C03648=1126.143,285.220,-74.172,-178.101,10.292,149.548
C03649=1126.148,284.972,-74.142,-178.104,10.290,149.548
C03650=1126.152,284.724,-74.112,-178.107,10.287,149.548
C03651=1126.156,284.475,-74.081,-178.109,10.284,149.548
C03652=1126.160,284.228,-74.051,-178.113,10.282,149.549
C03653=1126.165,283.980,-74.020,-178.116,10.279,149.549
C03654=1126.169,283.732,-73.989,-178.119,10.277,149.549
C03655=1126.173,283.483,-73.959,-178.122,10.274,149.549
C03656=1126.177,283.235,-73.928,-178.125,10.272,149.549
C03657=1126.181,282.988,-73.898,-178.128,10.269,149.549
C03658=1126.186,282.739,-73.868,-178.131,10.267,149.549
C03659=1126.189,282.491,-73.837,-178.134,10.265,149.550
C03660=1126.194,282.243,-73.807,-178.137,10.262,149.550
C03661=1126.199,281.995,-73.776,-178.140,10.259,149.550
C03662=1126.202,281.747,-73.746,-178.143,10.257,149.550
C03663=1126.207,281.498,-73.715,-178.146,10.254,149.550
C03664=1126.210,281.285,-73.689,-178.149,10.251,149.551
C03665=1126.214,281.072,-73.663,-178.152,10.249,149.551
C03666=1126.218,280.859,-73.638,-178.155,10.247,149.551
C03667=1126.221,280.645,-73.611,-178.158,10.244,149.551
C03668=1126.224,280.432,-73.585,-178.161,10.242,149.551
C03669=1126.228,280.218,-73.559,-178.164,10.239,149.551
C03670=1126.232,280.006,-73.533,-178.167,10.237,149.552
C03671=1126.235,279.791,-73.507,-178.170,10.235,149.552
C03672=1126.239,279.543,-73.477,-178.173,10.232,149.552
C03673=1126.244,279.295,-73.446,-178.177,10.229,149.552
C03674=1126.248,279.047,-73.417,-178.180,10.226,149.553
C03675=1126.253,278.799,-73.386,-178.183,10.224,149.553
C03676=1126.256,278.550,-73.356,-178.187,10.221,149.553
C03677=1126.260,278.303,-73.326,-178.190,10.218,149.553
C03678=1126.265,278.055,-73.295,-178.193,10.215,149.553
C03679=1126.269,277.806,-73.266,-178.196,10.212,149.553
C03680=1126.273,277.559,-73.236,-178.200,10.210,149.554
C03681=1126.278,277.310,-73.206,-178.203,10.207,149.554
C03682=1126.282,277.063,-73.175,-178.206,10.204,149.554
C03683=1126.285,276.814,-73.146,-178.210,10.201,149.554
C03684=1126.290,276.565,-73.115,-178.213,10.199,149.554
C03685=1126.294,276.317,-73.085,-178.215,10.196,149.554
C03686=1126.298,276.069,-73.056,-178.219,10.193,149.555
C03687=1126.302,275.821,-73.026,-178.222,10.191,149.555
C03688=1126.307,275.573,-72.996,-178.225,10.188,149.555
C03689=1126.311,275.325,-72.965,-178.228,10.185,149.555
C03690=1126.315,275.077,-72.936,-178.232,10.182,149.555
C03691=1126.319,274.829,-72.907,-178.235,10.179,149.555
C03692=1126.324,274.581,-72.876,-178.237,10.176,149.555
C03693=1126.328,274.332,-72.846,-178.241,10.174,149.556
C03694=1126.332,274.084,-72.817,-178.244,10.171,149.556
C03695=1126.335,273.836,-72.786,-178.247,10.168,149.556
C03696=1126.340,273.587,-72.756,-178.250,10.166,149.556
C03697=1126.345,273.339,-72.727,-178.253,10.163,149.556
C03698=1126.349,273.091,-72.697,-178.256,10.160,149.556
C03699=1126.353,272.843,-72.667,-178.258,10.159,149.556
C03700=1126.357,272.595,-72.638,-178.261,10.156,149.557
C03701=1126.361,272.347,-72.608,-178.264,10.153,149.557
C03702=1126.366,272.098,-72.578,-178.267,10.150,149.557
C03703=1126.370,271.850,-72.549,-178.270,10.148,149.557
C03704=1126.374,271.602,-72.519,-178.273,10.145,149.557
C03705=1126.378,271.354,-72.489,-178.276,10.142,149.557
C03706=1126.382,271.106,-72.460,-178.279,10.139,149.557
C03707=1126.387,270.857,-72.430,-178.281,10.137,149.557
C03708=1126.391,270.609,-72.401,-178.284,10.134,149.557
C03709=1126.395,270.361,-72.371,-178.287,10.132,149.558
C03710=1126.399,270.112,-72.342,-178.290,10.129,149.558
C03711=1126.403,269.864,-72.312,-178.292,10.127,149.558
C03712=1126.409,269.616,-72.283,-178.295,10.124,149.558
C03713=1126.413,269.368,-72.253,-178.298,10.121,149.558
C03714=1126.417,269.120,-72.223,-178.301,10.119,149.558
C03715=1126.421,268.872,-72.194,-178.303,10.117,149.558
C03716=1126.425,268.624,-72.164,-178.306,10.114,149.558
C03717=1126.429,268.376,-72.135,-178.309,10.111,149.558
C03718=1126.434,268.127,-72.105,-178.312,10.109,149.558
C03719=1126.438,267.879,-72.076,-178.314,10.106,149.559
C03720=1126.441,267.666,-72.051,-178.317,10.105,149.559
C03721=1126.445,267.452,-72.026,-178.319,10.102,149.559
C03722=1126.449,267.238,-72.001,-178.321,10.100,149.559
C03723=1126.452,267.025,-71.976,-178.323,10.098,149.559
C03724=1126.456,266.811,-71.951,-178.326,10.096,149.559
C03725=1126.460,266.598,-71.925,-178.328,10.094,149.559
C03726=1126.464,266.384,-71.900,-178.330,10.092,149.559
C03727=1126.467,266.171,-71.875,-178.332,10.090,149.559
C03728=1126.471,265.922,-71.845,-178.335,10.087,149.559
C03729=1126.476,265.674,-71.816,-178.337,10.085,149.559
C03730=1126.480,265.426,-71.786,-178.340,10.083,149.560
C03731=1126.484,265.178,-71.757,-178.343,10.080,149.560
C03732=1126.489,264.929,-71.728,-178.345,10.078,149.560
C03733=1126.492,264.681,-71.699,-178.347,10.075,149.560
C03734=1126.497,264.433,-71.670,-178.350,10.073,149.560
C03735=1126.501,264.185,-71.641,-178.354,10.070,149.560
C03736=1126.505,263.937,-71.611,-178.358,10.067,149.560
C03737=1126.510,263.688,-71.582,-178.362,10.064,149.561
C03738=1126.514,263.440,-71.553,-178.365,10.061,149.561
C03739=1126.518,263.191,-71.524,-178.369,10.058,149.561
C03740=1126.523,262.944,-71.494,-178.373,10.055,149.561
C03741=1126.527,262.695,-71.466,-178.376,10.052,149.561
C03742=1126.531,262.447,-71.437,-178.380,10.049,149.562
C03743=1126.535,262.199,-71.407,-178.383,10.045,149.562
C03744=1126.539,261.950,-71.379,-178.387,10.043,149.562
C03745=1126.544,261.702,-71.350,-178.390,10.039,149.562
C03746=1126.548,261.454,-71.321,-178.393,10.037,149.563
C03747=1126.552,261.205,-71.292,-178.397,10.033,149.563
C03748=1126.556,260.957,-71.263,-178.400,10.031,149.563
C03749=1126.561,260.709,-71.234,-178.404,10.027,149.563
C03750=1126.565,260.461,-71.205,-178.407,10.025,149.563
C03751=1126.569,260.212,-71.177,-178.410,10.021,149.563
C03752=1126.573,259.964,-71.147,-178.413,10.018,149.563
C03753=1126.579,259.716,-71.119,-178.416,10.016,149.563
C03754=1126.582,259.468,-71.090,-178.420,10.012,149.564
C03755=1126.586,259.219,-71.061,-178.423,10.010,149.564
C03756=1126.591,258.970,-71.032,-178.426,10.007,149.564
C03757=1126.595,258.723,-71.004,-178.429,10.004,149.564
C03758=1126.599,258.474,-70.974,-178.433,10.001,149.564
C03759=1126.604,258.225,-70.946,-178.436,9.998,149.564
C03760=1126.608,257.978,-70.918,-178.439,9.995,149.564
C03761=1126.612,257.729,-70.888,-178.442,9.992,149.564
C03762=1126.616,257.481,-70.860,-178.444,9.990,149.565
C03763=1126.621,257.233,-70.832,-178.448,9.986,149.564
C03764=1126.625,256.984,-70.802,-178.451,9.983,149.565
C03765=1126.629,256.736,-70.774,-178.454,9.980,149.565
C03766=1126.634,256.487,-70.746,-178.456,9.978,149.565
C03767=1126.638,256.240,-70.717,-178.459,9.975,149.565
C03768=1126.642,255.991,-70.688,-178.462,9.972,149.565
C03769=1126.646,255.743,-70.661,-178.462,9.971,149.565
C03770=1126.651,255.495,-70.631,-178.462,9.970,149.564
C03771=1126.655,255.246,-70.602,-178.462,9.969,149.564
C03772=1126.659,254.998,-70.575,-178.462,9.968,149.564
C03773=1126.664,254.749,-70.546,-178.462,9.967,149.564
C03774=1126.668,254.502,-70.517,-178.463,9.966,149.564
C03775=1126.672,254.253,-70.489,-178.464,9.964,149.563
C03776=1126.676,254.039,-70.464,-178.465,9.963,149.563
C03777=1126.679,253.826,-70.440,-178.466,9.962,149.563
C03778=1126.683,253.612,-70.415,-178.467,9.960,149.563
C03779=1126.687,253.397,-70.391,-178.468,9.959,149.563
C03780=1126.691,253.185,-70.366,-178.471,9.957,149.563
C03781=1126.694,252.971,-70.342,-178.472,9.955,149.563
C03782=1126.698,252.757,-70.318,-178.474,9.953,149.564
C03783=1126.702,252.544,-70.292,-178.476,9.951,149.564
C03784=1126.706,252.296,-70.265,-178.479,9.949,149.564
C03785=1126.710,252.047,-70.236,-178.482,9.946,149.564
C03786=1126.714,251.798,-70.208,-178.485,9.944,149.564
C03787=1126.719,251.550,-70.179,-178.488,9.941,149.564
C03788=1126.723,251.301,-70.151,-178.492,9.938,149.565
C03789=1126.728,251.054,-70.122,-178.495,9.936,149.565
C03790=1126.732,250.805,-70.094,-178.499,9.933,149.565
C03791=1126.736,250.556,-70.065,-178.504,9.929,149.566
C03792=1126.740,250.309,-70.037,-178.508,9.925,149.566
C03793=1126.745,250.060,-70.009,-178.513,9.922,149.566
C03794=1126.749,249.812,-69.981,-178.518,9.918,149.567
C03795=1126.753,249.563,-69.953,-178.523,9.914,149.567
C03796=1126.758,249.315,-69.924,-178.528,9.911,149.568
C03797=1126.762,249.066,-69.896,-178.533,9.906,149.568
C03798=1126.766,248.819,-69.868,-178.539,9.902,149.568
C03799=1126.771,248.570,-69.840,-178.545,9.896,149.569
C03800=1126.775,248.322,-69.812,-178.551,9.892,149.569
C03801=1126.779,248.073,-69.785,-178.557,9.887,149.570
C03802=1126.784,247.824,-69.756,-178.564,9.882,149.570
C03803=1126.788,247.576,-69.728,-178.570,9.877,149.571
C03804=1126.792,247.328,-69.700,-178.575,9.873,149.571
C03805=1126.796,247.079,-69.672,-178.576,9.870,149.571
C03806=1126.801,246.831,-69.645,-178.577,9.869,149.571
C03807=1126.806,246.583,-69.617,-178.579,9.866,149.570
C03808=1126.809,246.334,-69.589,-178.580,9.865,149.570
C03809=1126.814,246.086,-69.561,-178.582,9.862,149.570
C03810=1126.818,245.837,-69.533,-178.583,9.860,149.570
C03811=1126.822,245.589,-69.506,-178.585,9.858,149.570
C03812=1126.827,245.340,-69.477,-178.586,9.855,149.570
C03813=1126.831,245.092,-69.450,-178.588,9.853,149.570
C03814=1126.836,244.844,-69.422,-178.589,9.851,149.570
C03815=1126.839,244.595,-69.394,-178.591,9.849,149.570
C03816=1126.844,244.347,-69.367,-178.593,9.846,149.569
C03817=1126.849,244.098,-69.338,-178.595,9.844,149.569
C03818=1126.853,243.850,-69.310,-178.597,9.842,149.569
C03819=1126.858,243.602,-69.283,-178.598,9.839,149.569
C03820=1126.861,243.353,-69.255,-178.600,9.837,149.569
C03821=1126.866,243.105,-69.227,-178.602,9.836,149.569
C03822=1126.870,242.857,-69.200,-178.604,9.834,149.569
C03823=1126.874,242.608,-69.172,-178.606,9.831,149.569
C03824=1126.879,242.360,-69.145,-178.608,9.828,149.569
C03825=1126.883,242.111,-69.116,-178.610,9.826,149.569
C03826=1126.888,241.862,-69.089,-178.612,9.823,149.569
C03827=1126.892,241.614,-69.061,-178.614,9.821,149.569
C03828=1126.896,241.366,-69.033,-178.616,9.819,149.569
C03829=1126.901,241.117,-69.006,-178.618,9.817,149.569
C03830=1126.905,240.869,-68.978,-178.621,9.815,149.569
C03831=1126.909,240.620,-68.951,-178.623,9.812,149.569
C03832=1126.913,240.407,-68.928,-178.625,9.810,149.569
C03833=1126.917,240.192,-68.904,-178.627,9.808,149.569
C03834=1126.921,239.979,-68.880,-178.629,9.806,149.569
C03835=1126.924,239.766,-68.856,-178.631,9.804,149.569
C03836=1126.928,239.551,-68.833,-178.633,9.802,149.569
C03837=1126.932,239.338,-68.809,-178.635,9.800,149.569
C03838=1126.936,239.124,-68.785,-178.637,9.797,149.569
C03839=1126.940,238.910,-68.762,-178.639,9.795,149.569
C03840=1126.943,238.662,-68.734,-178.642,9.793,149.569
C03841=1126.948,238.413,-68.707,-178.644,9.790,149.569
C03842=1126.952,238.165,-68.679,-178.647,9.787,149.570
C03843=1126.957,237.916,-68.651,-178.649,9.785,149.570
C03844=1126.961,237.668,-68.624,-178.652,9.783,149.570
C03845=1126.966,237.420,-68.597,-178.655,9.780,149.570
C03846=1126.970,237.171,-68.570,-178.657,9.778,149.570
C03847=1126.974,236.922,-68.542,-178.660,9.775,149.570
C03848=1126.979,236.674,-68.514,-178.663,9.772,149.570
C03849=1126.983,236.426,-68.487,-178.666,9.769,149.570
C03850=1126.987,236.177,-68.460,-178.669,9.767,149.570
C03851=1126.991,235.929,-68.433,-178.672,9.764,149.570
C03852=1126.996,235.681,-68.406,-178.674,9.761,149.570
C03853=1127.000,235.432,-68.379,-178.677,9.758,149.571
C03854=1127.005,235.184,-68.352,-178.680,9.755,149.571
C03855=1127.009,234.935,-68.323,-178.683,9.753,149.571
C03856=1127.013,234.686,-68.296,-178.686,9.750,149.571
C03857=1127.018,234.438,-68.269,-178.689,9.747,149.571
C03858=1127.022,234.190,-68.243,-178.692,9.744,149.571
C03859=1127.026,233.941,-68.215,-178.695,9.742,149.571
C03860=1127.030,233.693,-68.188,-178.699,9.738,149.572
C03861=1127.035,233.444,-68.161,-178.702,9.736,149.572
C03862=1127.040,233.196,-68.133,-178.705,9.733,149.572
C03863=1127.044,232.947,-68.106,-178.709,9.729,149.572
C03864=1127.048,232.699,-68.080,-178.711,9.727,149.572
C03865=1127.052,232.450,-68.053,-178.714,9.724,149.572
C03866=1127.057,232.201,-68.025,-178.718,9.720,149.572
C03867=1127.062,231.953,-67.998,-178.721,9.718,149.572
C03868=1127.065,231.705,-67.972,-178.725,9.714,149.573
C03869=1127.070,231.456,-67.945,-178.728,9.711,149.573
C03870=1127.075,231.208,-67.918,-178.731,9.708,149.573
C03871=1127.079,230.959,-67.891,-178.735,9.705,149.573
C03872=1127.083,230.710,-67.864,-178.739,9.701,149.573
C03873=1127.087,230.462,-67.837,-178.742,9.698,149.573
C03874=1127.092,230.213,-67.810,-178.745,9.695,149.573
C03875=1127.096,229.965,-67.783,-178.749,9.691,149.574
C03876=1127.101,229.717,-67.756,-178.753,9.688,149.574
C03877=1127.105,229.468,-67.729,-178.756,9.685,149.574
C03878=1127.109,229.220,-67.703,-178.760,9.681,149.574
C03879=1127.114,228.971,-67.676,-178.763,9.678,149.574
C03880=1127.119,228.722,-67.649,-178.767,9.674,149.574
C03881=1127.123,228.474,-67.623,-178.771,9.671,149.574
C03882=1127.127,228.226,-67.596,-178.774,9.667,149.575
C03883=1127.131,227.977,-67.569,-178.777,9.664,149.575
C03884=1127.136,227.728,-67.543,-178.781,9.661,149.575
C03885=1127.140,227.479,-67.516,-178.784,9.657,149.575
C03886=1127.144,227.231,-67.489,-178.788,9.653,149.575
C03887=1127.149,226.982,-67.462,-178.790,9.651,149.575
C03888=1127.153,226.769,-67.439,-178.793,9.648,149.575
C03889=1127.157,226.555,-67.416,-178.796,9.645,149.575
C03890=1127.160,226.341,-67.393,-178.799,9.642,149.575
C03891=1127.164,226.127,-67.371,-178.801,9.639,149.575
C03892=1127.168,225.913,-67.349,-178.804,9.636,149.575
C03893=1127.172,225.699,-67.326,-178.807,9.633,149.575
C03894=1127.176,225.485,-67.303,-178.810,9.630,149.575
C03895=1127.180,225.272,-67.280,-178.812,9.627,149.575
C03896=1127.184,225.023,-67.253,-178.816,9.624,149.575
C03897=1127.188,224.774,-67.227,-178.818,9.621,149.575
C03898=1127.192,224.526,-67.201,-178.822,9.617,149.575
C03899=1127.197,224.278,-67.174,-178.825,9.614,149.575
C03900=1127.201,224.029,-67.148,-178.827,9.611,149.575
C03901=1127.206,223.780,-67.121,-178.831,9.607,149.575
C03902=1127.210,223.531,-67.095,-178.833,9.604,149.575
C03903=1127.215,223.283,-67.068,-178.836,9.600,149.575
C03904=1127.219,223.034,-67.043,-178.839,9.597,149.575
C03905=1127.223,222.786,-67.016,-178.842,9.595,149.575
C03906=1127.228,222.537,-66.990,-178.844,9.591,149.575
C03907=1127.232,222.288,-66.964,-178.848,9.588,149.575
C03908=1127.237,222.041,-66.938,-178.850,9.584,149.575
C03909=1127.242,221.791,-66.912,-178.853,9.581,149.575
C03910=1127.246,221.543,-66.885,-178.855,9.578,149.575
C03911=1127.251,221.294,-66.859,-178.858,9.575,149.575
C03912=1127.255,221.045,-66.833,-178.860,9.572,149.575
C03913=1127.259,220.797,-66.807,-178.863,9.568,149.575
C03914=1127.263,220.548,-66.781,-178.866,9.565,149.575
C03915=1127.268,220.300,-66.755,-178.868,9.562,149.575
C03916=1127.272,220.052,-66.728,-178.871,9.559,149.575
C03917=1127.277,219.803,-66.703,-178.873,9.556,149.575
C03918=1127.282,219.554,-66.676,-178.876,9.553,149.575
C03919=1127.285,219.306,-66.650,-178.878,9.550,149.574
C03920=1127.290,219.057,-66.624,-178.880,9.547,149.574
C03921=1127.294,218.808,-66.598,-178.883,9.544,149.574
C03922=1127.299,218.560,-66.572,-178.885,9.541,149.574
C03923=1127.303,218.311,-66.546,-178.888,9.537,149.574
C03924=1127.308,218.063,-66.520,-178.890,9.534,149.574
C03925=1127.312,217.814,-66.494,-178.892,9.532,149.574
C03926=1127.316,217.565,-66.469,-178.894,9.529,149.574
C03927=1127.322,217.317,-66.443,-178.897,9.525,149.574
C03928=1127.326,217.068,-66.416,-178.898,9.523,149.573
C03929=1127.330,216.820,-66.390,-178.901,9.520,149.573
C03930=1127.334,216.571,-66.365,-178.903,9.516,149.573
C03931=1127.338,216.322,-66.339,-178.905,9.514,149.573
C03932=1127.343,216.074,-66.313,-178.907,9.511,149.573
C03933=1127.348,215.825,-66.287,-178.909,9.508,149.573
C03934=1127.352,215.576,-66.261,-178.911,9.505,149.573
C03935=1127.356,215.327,-66.236,-178.913,9.503,149.573
C03936=1127.361,215.079,-66.210,-178.915,9.500,149.572
C03937=1127.366,214.830,-66.184,-178.917,9.497,149.572
C03938=1127.369,214.582,-66.158,-178.919,9.494,149.572
C03939=1127.374,214.333,-66.132,-178.921,9.491,149.572
C03940=1127.378,214.085,-66.107,-178.923,9.488,149.572
C03941=1127.383,213.836,-66.081,-178.924,9.486,149.572
C03942=1127.388,213.587,-66.055,-178.926,9.484,149.572
C03943=1127.392,213.338,-66.029,-178.928,9.481,149.571
C03944=1127.396,213.124,-66.008,-178.930,9.479,149.571
C03945=1127.400,212.910,-65.985,-178.931,9.476,149.571
C03946=1127.403,212.697,-65.963,-178.932,9.474,149.571
C03947=1127.407,212.483,-65.941,-178.934,9.472,149.571
C03948=1127.411,212.269,-65.920,-178.936,9.469,149.571
C03949=1127.415,212.055,-65.897,-178.938,9.467,149.571
C03950=1127.418,211.840,-65.875,-178.939,9.465,149.571
C03951=1127.423,211.626,-65.853,-178.940,9.463,149.570
C03952=1127.427,211.378,-65.828,-178.942,9.460,149.570
C03953=1127.432,211.129,-65.802,-178.945,9.457,149.570
C03954=1127.436,210.880,-65.776,-178.947,9.455,149.570
C03955=1127.441,210.632,-65.751,-178.949,9.453,149.570
C03956=1127.445,210.383,-65.725,-178.951,9.449,149.570
C03957=1127.449,210.135,-65.699,-178.953,9.447,149.570
C03958=1127.454,209.886,-65.675,-178.955,9.445,149.570
C03959=1127.458,209.637,-65.649,-178.957,9.442,149.570
C03960=1127.463,209.388,-65.623,-178.959,9.439,149.570
C03961=1127.467,209.140,-65.598,-178.962,9.436,149.570
C03962=1127.472,208.891,-65.572,-178.964,9.434,149.570
C03963=1127.476,208.643,-65.546,-178.967,9.431,149.570
C03964=1127.481,208.394,-65.522,-178.969,9.428,149.570
C03965=1127.485,208.145,-65.496,-178.972,9.426,149.570
C03966=1127.489,207.896,-65.470,-178.974,9.423,149.570
C03967=1127.494,207.648,-65.445,-178.977,9.420,149.570
C03968=1127.499,207.399,-65.420,-178.979,9.418,149.570
C03969=1127.503,207.151,-65.395,-178.981,9.415,149.570
C03970=1127.507,206.902,-65.369,-178.984,9.412,149.570
C03971=1127.511,206.653,-65.343,-178.987,9.409,149.570
C03972=1127.517,206.405,-65.319,-178.989,9.407,149.570
C03973=1127.521,206.156,-65.293,-178.992,9.404,149.571
C03974=1127.526,205.908,-65.268,-178.995,9.401,149.571
C03975=1127.530,205.658,-65.242,-178.998,9.398,149.571
C03976=1127.535,205.410,-65.217,-179.001,9.396,149.571
C03977=1127.539,205.161,-65.193,-179.003,9.393,149.571
C03978=1127.543,204.912,-65.167,-179.006,9.390,149.571
C03979=1127.548,204.664,-65.142,-179.009,9.387,149.571
C03980=1127.552,204.415,-65.116,-179.012,9.384,149.571
C03981=1127.557,204.167,-65.091,-179.016,9.381,149.571
C03982=1127.562,203.917,-65.066,-179.018,9.378,149.571
C03983=1127.566,203.669,-65.041,-179.021,9.375,149.571
C03984=1127.570,203.420,-65.016,-179.024,9.372,149.572
C03985=1127.575,203.172,-64.991,-179.028,9.369,149.572
C03986=1127.580,202.922,-64.966,-179.031,9.366,149.572
C03987=1127.584,202.675,-64.941,-179.034,9.363,149.572
C03988=1127.588,202.425,-64.916,-179.037,9.360,149.572
C03989=1127.593,202.177,-64.891,-179.040,9.357,149.572
C03990=1127.597,201.928,-64.866,-179.044,9.353,149.572
C03991=1127.602,201.680,-64.841,-179.046,9.350,149.572
C03992=1127.606,201.430,-64.816,-179.050,9.347,149.573
C03993=1127.611,201.182,-64.792,-179.053,9.344,149.573
C03994=1127.615,200.933,-64.766,-179.056,9.341,149.573
C03995=1127.620,200.685,-64.741,-179.060,9.337,149.573
C03996=1127.623,200.436,-64.716,-179.063,9.334,149.573
C03997=1127.629,200.187,-64.691,-179.066,9.331,149.573
C03998=1127.633,199.938,-64.666,-179.070,9.327,149.573
C03999=1127.638,199.689,-64.642,-179.074,9.324,149.573
C04000=1127.641,199.476,-64.621,-179.077,9.321,149.574
C04001=1127.645,199.261,-64.599,-179.080,9.318,149.574
C04002=1127.649,199.047,-64.577,-179.083,9.315,149.574
C04003=1127.653,198.833,-64.557,-179.086,9.312,149.574
C04004=1127.657,198.619,-64.535,-179.089,9.309,149.574
C04005=1127.661,198.405,-64.515,-179.093,9.306,149.574
C04006=1127.665,198.191,-64.493,-179.095,9.303,149.574
C04007=1127.668,197.977,-64.472,-179.099,9.299,149.574
C04008=1127.673,197.728,-64.447,-179.102,9.296,149.575
C04009=1127.677,197.479,-64.423,-179.106,9.292,149.575
C04010=1127.682,197.230,-64.398,-179.109,9.289,149.575
C04011=1127.686,196.981,-64.373,-179.114,9.284,149.575
C04012=1127.691,196.733,-64.349,-179.117,9.281,149.575
C04013=1127.696,196.484,-64.325,-179.121,9.277,149.575
C04014=1127.700,196.235,-64.300,-179.125,9.273,149.575
C04015=1127.705,195.986,-64.276,-179.126,9.271,149.575
C04016=1127.710,195.738,-64.251,-179.127,9.268,149.575
C04017=1127.713,195.489,-64.226,-179.129,9.266,149.575
C04018=1127.718,195.240,-64.201,-179.131,9.263,149.575
C04019=1127.723,194.992,-64.177,-179.132,9.261,149.574
C04020=1127.727,194.743,-64.153,-179.134,9.258,149.574
C04021=1127.732,194.493,-64.129,-179.136,9.256,149.574
C04022=1127.736,194.245,-64.105,-179.137,9.253,149.574
C04023=1127.742,193.996,-64.080,-179.139,9.251,149.574
C04024=1127.745,193.747,-64.055,-179.141,9.248,149.574
C04025=1127.750,193.499,-64.031,-179.142,9.246,149.574
C04026=1127.755,193.250,-64.007,-179.145,9.242,149.574
C04027=1127.759,193.001,-63.982,-179.146,9.240,149.573
C04028=1127.764,192.752,-63.958,-179.148,9.237,149.573
C04029=1127.768,192.504,-63.934,-179.150,9.235,149.573
C04030=1127.773,192.255,-63.909,-179.151,9.232,149.573
C04031=1127.777,192.006,-63.884,-179.154,9.229,149.573
C04032=1127.781,191.758,-63.860,-179.156,9.227,149.573
C04033=1127.786,191.509,-63.837,-179.158,9.225,149.573
C04034=1127.791,191.260,-63.812,-179.159,9.222,149.573
C04035=1127.795,191.011,-63.788,-179.162,9.219,149.573
C04036=1127.800,190.762,-63.764,-179.164,9.217,149.573
C04037=1127.805,190.514,-63.739,-179.166,9.214,149.573
C04038=1127.809,190.265,-63.715,-179.168,9.211,149.573
C04039=1127.813,190.015,-63.691,-179.170,9.208,149.572
C04040=1127.818,189.767,-63.667,-179.172,9.205,149.572
C04041=1127.823,189.518,-63.643,-179.174,9.203,149.572
C04042=1127.827,189.270,-63.619,-179.177,9.200,149.572
C04043=1127.832,189.021,-63.595,-179.178,9.198,149.572
C04044=1127.836,188.771,-63.570,-179.181,9.194,149.572
C04045=1127.841,188.523,-63.546,-179.183,9.192,149.572
C04046=1127.845,188.275,-63.522,-179.185,9.189,149.572
C04047=1127.850,188.026,-63.499,-179.188,9.186,149.572
C04048=1127.854,187.777,-63.475,-179.190,9.184,149.572
C04049=1127.859,187.528,-63.450,-179.192,9.180,149.572
C04050=1127.863,187.279,-63.426,-179.195,9.177,149.572
C04051=1127.868,187.030,-63.402,-179.197,9.175,149.572
C04052=1127.872,186.782,-63.378,-179.200,9.172,149.572
C04053=1127.877,186.533,-63.355,-179.202,9.169,149.572
C04054=1127.882,186.284,-63.330,-179.205,9.166,149.572
C04055=1127.886,186.036,-63.306,-179.207,9.163,149.572
C04056=1127.890,185.821,-63.285,-179.209,9.161,149.572
C04057=1127.894,185.607,-63.265,-179.211,9.158,149.572
C04058=1127.897,185.392,-63.244,-179.214,9.155,149.572
C04059=1127.902,185.178,-63.224,-179.215,9.153,149.572
C04060=1127.906,184.964,-63.203,-179.218,9.151,149.572
C04061=1127.910,184.749,-63.182,-179.220,9.148,149.572
C04062=1127.914,184.536,-63.162,-179.222,9.145,149.572
C04063=1127.917,184.321,-63.142,-179.225,9.142,149.572
C04064=1127.922,184.073,-63.118,-179.227,9.139,149.572
C04065=1127.927,183.824,-63.094,-179.230,9.136,149.572
C04066=1127.931,183.575,-63.071,-179.233,9.133,149.572
C04067=1127.936,183.326,-63.047,-179.235,9.130,149.572
C04068=1127.940,183.077,-63.023,-179.238,9.127,149.572
C04069=1127.945,182.829,-62.999,-179.241,9.124,149.572
C04070=1127.950,182.579,-62.975,-179.244,9.121,149.572
C04071=1127.954,182.330,-62.951,-179.246,9.117,149.572
C04072=1127.959,182.081,-62.928,-179.249,9.115,149.572
C04073=1127.963,181.832,-62.904,-179.253,9.111,149.572
C04074=1127.968,181.584,-62.880,-179.255,9.108,149.572
C04075=1127.972,181.335,-62.857,-179.258,9.105,149.572
C04076=1127.977,181.086,-62.834,-179.261,9.101,149.572
C04077=1127.981,180.838,-62.810,-179.264,9.098,149.572
C04078=1127.986,180.589,-62.787,-179.267,9.094,149.572
C04079=1127.990,180.340,-62.763,-179.270,9.091,149.572
C04080=1127.995,180.091,-62.739,-179.273,9.087,149.572
C04081=1127.999,179.842,-62.716,-179.275,9.084,149.572
C04082=1128.004,179.593,-62.693,-179.279,9.081,149.572
C04083=1128.009,179.344,-62.669,-179.282,9.078,149.572
C04084=1128.013,179.096,-62.645,-179.284,9.075,149.572
C04085=1128.018,178.847,-62.622,-179.287,9.072,149.572
C04086=1128.023,178.598,-62.598,-179.289,9.068,149.572
C04087=1128.027,178.349,-62.575,-179.291,9.066,149.572
C04088=1128.032,178.100,-62.552,-179.293,9.062,149.571
C04089=1128.036,177.851,-62.528,-179.295,9.060,149.571
C04090=1128.040,177.602,-62.505,-179.297,9.057,149.571
C04091=1128.045,177.353,-62.481,-179.299,9.053,149.571
C04092=1128.050,177.104,-62.458,-179.301,9.051,149.571
C04093=1128.054,176.855,-62.435,-179.304,9.048,149.571
C04094=1128.059,176.606,-62.411,-179.306,9.044,149.571
C04095=1128.064,176.358,-62.389,-179.308,9.042,149.571
C04096=1128.068,176.109,-62.366,-179.310,9.039,149.571
C04097=1128.073,175.860,-62.342,-179.312,9.035,149.571
C04098=1128.077,175.612,-62.318,-179.314,9.033,149.571
C04099=1128.082,175.363,-62.295,-179.317,9.030,149.571
C04100=1128.086,175.114,-62.272,-179.319,9.027,149.570
C04101=1128.091,174.865,-62.249,-179.321,9.024,149.570
C04102=1128.095,174.616,-62.225,-179.323,9.021,149.570
C04103=1128.100,174.367,-62.202,-179.326,9.018,149.570
C04104=1128.104,174.118,-62.179,-179.327,9.015,149.570
C04105=1128.109,173.870,-62.156,-179.330,9.012,149.570
C04106=1128.114,173.621,-62.133,-179.332,9.009,149.570
C04107=1128.119,173.372,-62.110,-179.335,9.006,149.570
C04108=1128.123,173.122,-62.087,-179.336,9.003,149.570
C04109=1128.128,172.873,-62.064,-179.339,9.000,149.570
C04110=1128.133,172.624,-62.041,-179.341,8.997,149.570
C04111=1128.136,172.376,-62.018,-179.343,8.994,149.569
C04112=1128.141,172.162,-61.998,-179.345,8.991,149.569
C04113=1128.144,171.947,-61.978,-179.347,8.989,149.569
C04114=1128.149,171.733,-61.958,-179.349,8.987,149.569
C04115=1128.152,171.518,-61.938,-179.351,8.983,149.569
C04116=1128.157,171.304,-61.919,-179.353,8.981,149.569
C04117=1128.161,171.090,-61.899,-179.355,8.978,149.569
C04118=1128.165,170.875,-61.879,-179.357,8.976,149.569
C04119=1128.169,170.661,-61.859,-179.359,8.973,149.569
C04120=1128.173,170.412,-61.837,-179.361,8.970,149.569
C04121=1128.178,170.163,-61.814,-179.363,8.967,149.569
C04122=1128.183,169.914,-61.790,-179.366,8.964,149.569
C04123=1128.187,169.665,-61.767,-179.368,8.961,149.568
C04124=1128.192,169.417,-61.744,-179.370,8.958,149.568
C04125=1128.196,169.167,-61.722,-179.373,8.954,149.568
C04126=1128.201,168.918,-61.699,-179.376,8.951,149.568
C04127=1128.206,168.669,-61.676,-179.377,8.949,149.568
C04128=1128.211,168.421,-61.654,-179.379,8.945,149.568
C04129=1128.215,168.172,-61.631,-179.382,8.942,149.568
C04130=1128.219,167.923,-61.608,-179.385,8.939,149.568
C04131=1128.224,167.673,-61.585,-179.387,8.936,149.568
C04132=1128.229,167.425,-61.563,-179.389,8.933,149.568
C04133=1128.233,167.176,-61.539,-179.392,8.930,149.568
C04134=1128.238,166.927,-61.517,-179.394,8.926,149.568
C04135=1128.242,166.678,-61.494,-179.397,8.923,149.567
C04136=1128.247,166.430,-61.472,-179.399,8.920,149.567
C04137=1128.252,166.180,-61.449,-179.401,8.917,149.567
C04138=1128.256,165.932,-61.426,-179.404,8.914,149.567
C04139=1128.262,165.683,-61.404,-179.406,8.911,149.567
C04140=1128.266,165.434,-61.381,-179.408,8.908,149.567
C04141=1128.271,165.184,-61.359,-179.410,8.905,149.567
C04142=1128.275,164.936,-61.336,-179.413,8.902,149.567
C04143=1128.280,164.687,-61.313,-179.415,8.899,149.567
C04144=1128.284,164.438,-61.291,-179.417,8.895,149.567
C04145=1128.289,164.189,-61.267,-179.420,8.892,149.567
C04146=1128.294,163.940,-61.246,-179.423,8.888,149.567
C04147=1128.298,163.691,-61.224,-179.426,8.885,149.566
C04148=1128.303,163.442,-61.200,-179.428,8.881,149.566
C04149=1128.307,163.193,-61.179,-179.430,8.878,149.566
C04150=1128.311,162.944,-61.156,-179.433,8.875,149.566
C04151=1128.316,162.695,-61.133,-179.435,8.872,149.566
C04152=1128.321,162.447,-61.111,-179.437,8.869,149.566
C04153=1128.326,162.197,-61.088,-179.440,8.866,149.566
C04154=1128.331,161.948,-61.066,-179.442,8.862,149.566
C04155=1128.335,161.700,-61.044,-179.445,8.859,149.566
C04156=1128.340,161.450,-61.021,-179.447,8.856,149.566
C04157=1128.345,161.201,-60.999,-179.450,8.853,149.566
C04158=1128.349,160.953,-60.977,-179.452,8.848,149.565
C04159=1128.354,160.704,-60.955,-179.455,8.845,149.565
C04160=1128.359,160.454,-60.932,-179.457,8.842,149.565
C04161=1128.363,160.206,-60.910,-179.460,8.839,149.565
C04162=1128.367,159.957,-60.888,-179.462,8.836,149.565
C04163=1128.372,159.707,-60.865,-179.465,8.833,149.565
C04164=1128.377,159.459,-60.844,-179.468,8.829,149.565
C04165=1128.381,159.210,-60.821,-179.470,8.825,149.565
C04166=1128.386,158.961,-60.799,-179.472,8.822,149.565
C04167=1128.391,158.712,-60.776,-179.475,8.819,149.565
C04168=1128.395,158.498,-60.757,-179.477,8.815,149.564
C04169=1128.399,158.283,-60.738,-179.479,8.812,149.564
C04170=1128.403,158.068,-60.719,-179.481,8.810,149.564
C04171=1128.407,157.854,-60.700,-179.483,8.807,149.564
C04172=1128.411,157.639,-60.681,-179.486,8.803,149.564
C04173=1128.415,157.425,-60.662,-179.488,8.801,149.564
C04174=1128.419,157.210,-60.643,-179.490,8.798,149.564
C04175=1128.423,156.996,-60.624,-179.492,8.795,149.564
C04176=1128.428,156.748,-60.602,-179.495,8.791,149.564
C04177=1128.432,156.498,-60.580,-179.497,8.788,149.564
C04178=1128.437,156.250,-60.558,-179.500,8.784,149.563
C04179=1128.441,156.000,-60.536,-179.503,8.781,149.563
C04180=1128.446,155.752,-60.515,-179.505,8.777,149.563
C04181=1128.450,155.502,-60.493,-179.508,8.774,149.563
C04182=1128.455,155.254,-60.471,-179.510,8.770,149.563
C04183=1128.460,155.004,-60.448,-179.513,8.767,149.563
C04184=1128.465,154.755,-60.427,-179.516,8.763,149.563
C04185=1128.469,154.506,-60.404,-179.518,8.760,149.563
C04186=1128.474,154.257,-60.383,-179.520,8.756,149.563
C04187=1128.478,154.008,-60.361,-179.523,8.752,149.562
C04188=1128.483,153.759,-60.339,-179.526,8.749,149.562
C04189=1128.488,153.511,-60.317,-179.528,8.745,149.562
C04190=1128.493,153.261,-60.296,-179.531,8.742,149.562
C04191=1128.498,153.012,-60.274,-179.533,8.737,149.562
C04192=1128.502,152.763,-60.252,-179.536,8.734,149.562
C04193=1128.507,152.514,-60.231,-179.539,8.730,149.562
C04194=1128.512,152.266,-60.209,-179.541,8.727,149.562
C04195=1128.516,152.016,-60.187,-179.544,8.723,149.561
C04196=1128.521,151.768,-60.165,-179.546,8.720,149.561
C04197=1128.525,151.518,-60.144,-179.549,8.715,149.561
C04198=1128.530,151.269,-60.122,-179.552,8.712,149.561
C04199=1128.535,151.020,-60.101,-179.554,8.708,149.561
C04200=1128.539,150.771,-60.078,-179.557,8.705,149.561
C04201=1128.545,150.522,-60.058,-179.560,8.701,149.561
C04202=1128.549,150.273,-60.036,-179.562,8.698,149.561
C04203=1128.554,150.024,-60.014,-179.565,8.693,149.560
C04204=1128.559,149.775,-59.992,-179.568,8.689,149.560
C04205=1128.563,149.526,-59.972,-179.570,8.686,149.560
C04206=1128.567,149.277,-59.950,-179.573,8.682,149.560
C04207=1128.572,149.028,-59.928,-179.575,8.679,149.560
C04208=1128.577,148.779,-59.907,-179.578,8.674,149.560
C04209=1128.582,148.530,-59.885,-179.581,8.670,149.559
C04210=1128.587,148.280,-59.864,-179.583,8.667,149.559
C04211=1128.592,148.032,-59.842,-179.586,8.663,149.559
C04212=1128.596,147.783,-59.821,-179.589,8.658,149.559
C04213=1128.600,147.533,-59.800,-179.591,8.655,149.559
C04214=1128.605,147.285,-59.778,-179.594,8.651,149.559
C04215=1128.610,147.035,-59.757,-179.597,8.647,149.558
C04216=1128.615,146.786,-59.735,-179.600,8.643,149.558
C04217=1128.619,146.537,-59.715,-179.602,8.639,149.558
C04218=1128.624,146.289,-59.693,-179.605,8.635,149.558
C04219=1128.629,146.039,-59.672,-179.608,8.631,149.558
C04220=1128.634,145.791,-59.651,-179.610,8.627,149.558
C04221=1128.638,145.541,-59.630,-179.613,8.623,149.557
C04222=1128.643,145.292,-59.608,-179.615,8.619,149.557
C04223=1128.648,145.043,-59.587,-179.618,8.615,149.557
C04224=1128.651,144.829,-59.569,-179.619,8.612,149.557
C04225=1128.656,144.614,-59.551,-179.621,8.609,149.556
C04226=1128.660,144.400,-59.532,-179.622,8.606,149.556
C04227=1128.664,144.185,-59.514,-179.623,8.604,149.556
C04228=1128.668,143.970,-59.496,-179.624,8.601,149.555
C04229=1128.672,143.756,-59.478,-179.626,8.598,149.555
C04230=1128.676,143.541,-59.460,-179.627,8.595,149.555
C04231=1128.680,143.326,-59.442,-179.628,8.592,149.554
C04232=1128.685,143.077,-59.421,-179.629,8.589,149.554
C04233=1128.690,142.829,-59.399,-179.631,8.585,149.554
C04234=1128.694,142.579,-59.378,-179.632,8.582,149.553
C04235=1128.699,142.330,-59.357,-179.634,8.579,149.553
C04236=1128.704,142.081,-59.336,-179.635,8.576,149.553
C04237=1128.708,141.832,-59.315,-179.636,8.573,149.552
C04238=1128.713,141.583,-59.294,-179.639,8.569,149.552
C04239=1128.717,141.334,-59.273,-179.640,8.566,149.552
C04240=1128.722,141.085,-59.252,-179.642,8.563,149.551
C04241=1128.727,140.835,-59.231,-179.643,8.560,149.551
C04242=1128.732,140.586,-59.211,-179.645,8.556,149.551
C04243=1128.736,140.338,-59.189,-179.646,8.553,149.550
C04244=1128.741,140.089,-59.169,-179.647,8.549,149.550
C04245=1128.746,139.839,-59.148,-179.649,8.546,149.550
C04246=1128.750,139.591,-59.127,-179.650,8.543,149.549
C04247=1128.756,139.341,-59.106,-179.652,8.540,149.549
C04248=1128.760,139.092,-59.084,-179.654,8.536,149.549
C04249=1128.764,138.843,-59.064,-179.655,8.533,149.548
C04250=1128.770,138.594,-59.043,-179.657,8.529,149.548
C04251=1128.774,138.345,-59.023,-179.658,8.527,149.548
C04252=1128.779,138.095,-59.002,-179.660,8.523,149.547
C04253=1128.784,137.847,-58.981,-179.661,8.520,149.547
C04254=1128.789,137.597,-58.960,-179.663,8.517,149.547
C04255=1128.793,137.348,-58.940,-179.664,8.513,149.546
C04256=1128.798,137.100,-58.918,-179.666,8.510,149.546
C04257=1128.803,136.851,-58.898,-179.667,8.507,149.546
C04258=1128.808,136.601,-58.877,-179.669,8.503,149.545
C04259=1128.812,136.353,-58.856,-179.670,8.500,149.545
C04260=1128.817,136.104,-58.836,-179.672,8.497,149.545
C04261=1128.821,135.854,-58.815,-179.673,8.494,149.544
C04262=1128.826,135.605,-58.794,-179.676,8.490,149.544
C04263=1128.831,135.355,-58.773,-179.677,8.488,149.544
C04264=1128.835,135.106,-58.753,-179.679,8.484,149.543
C04265=1128.840,134.857,-58.732,-179.680,8.481,149.543
C04266=1128.845,134.608,-58.712,-179.682,8.477,149.543
C04267=1128.850,134.359,-58.691,-179.684,8.474,149.543
C04268=1128.854,134.110,-58.670,-179.685,8.471,149.542
C04269=1128.859,133.861,-58.650,-179.687,8.467,149.542
C04270=1128.864,133.612,-58.629,-179.688,8.464,149.542
C04271=1128.868,133.363,-58.609,-179.690,8.461,149.542
C04272=1128.874,133.114,-58.588,-179.691,8.458,149.541
C04273=1128.878,132.865,-58.567,-179.693,8.454,149.541
C04274=1128.883,132.616,-58.547,-179.696,8.451,149.541
C04275=1128.888,132.366,-58.527,-179.697,8.448,149.540
C04276=1128.892,132.117,-58.506,-179.699,8.444,149.540
C04277=1128.897,131.868,-58.486,-179.700,8.441,149.540
C04278=1128.902,131.619,-58.465,-179.702,8.438,149.539
C04279=1128.906,131.370,-58.445,-179.704,8.434,149.539
C04280=1128.911,131.156,-58.427,-179.705,8.431,149.539
C04281=1128.915,130.941,-58.410,-179.707,8.429,149.539
C04282=1128.919,130.726,-58.392,-179.708,8.426,149.538
C04283=1128.923,130.511,-58.375,-179.709,8.423,149.538
C04284=1128.927,130.296,-58.357,-179.711,8.420,149.538
C04285=1128.932,130.082,-58.339,-179.712,8.417,149.538
C04286=1128.936,129.867,-58.322,-179.713,8.415,149.537
C04287=1128.939,129.653,-58.304,-179.715,8.412,149.537
C04288=1128.944,129.404,-58.284,-179.717,8.408,149.537
C04289=1128.949,129.154,-58.264,-179.719,8.405,149.536
C04290=1128.954,128.905,-58.243,-179.720,8.402,149.536
C04291=1128.958,128.656,-58.223,-179.722,8.398,149.536
C04292=1128.963,128.406,-58.203,-179.724,8.395,149.536
C04293=1128.969,128.158,-58.183,-179.725,8.392,149.535
C04294=1128.973,127.909,-58.162,-179.727,8.388,149.535
C04295=1128.977,127.660,-58.142,-179.729,8.385,149.535
C04296=1128.982,127.410,-58.122,-179.731,8.382,149.535
C04297=1128.987,127.161,-58.101,-179.732,8.378,149.534
C04298=1128.992,126.912,-58.081,-179.734,8.375,149.534
C04299=1128.997,126.663,-58.061,-179.736,8.372,149.534
C04300=1129.001,126.414,-58.041,-179.738,8.369,149.534
C04301=1129.005,126.165,-58.020,-179.740,8.365,149.533
C04302=1129.011,125.916,-58.001,-179.741,8.362,149.533
C04303=1129.016,125.667,-57.980,-179.743,8.358,149.533
C04304=1129.021,125.417,-57.960,-179.745,8.355,149.532
C04305=1129.025,125.168,-57.940,-179.746,8.352,149.532
C04306=1129.030,124.919,-57.920,-179.748,8.348,149.532
C04307=1129.034,124.670,-57.900,-179.750,8.345,149.532
C04308=1129.039,124.421,-57.880,-179.752,8.341,149.531
C04309=1129.044,124.172,-57.860,-179.754,8.339,149.531
C04310=1129.049,123.923,-57.840,-179.755,8.335,149.531
C04311=1129.053,123.673,-57.820,-179.757,8.331,149.530
C04312=1129.058,123.424,-57.799,-179.759,8.329,149.530
C04313=1129.063,123.174,-57.780,-179.761,8.325,149.530
C04314=1129.068,122.926,-57.760,-179.763,8.322,149.530
C04315=1129.073,122.677,-57.740,-179.765,8.318,149.529
C04316=1129.077,122.428,-57.720,-179.766,8.315,149.529
C04317=1129.082,122.178,-57.700,-179.768,8.311,149.529
C04318=1129.087,121.929,-57.680,-179.770,8.308,149.529
C04319=1129.092,121.680,-57.660,-179.772,8.304,149.529
C04320=1129.097,121.431,-57.641,-179.773,8.301,149.528
C04321=1129.101,121.182,-57.620,-179.775,8.298,149.528
C04322=1129.106,120.932,-57.601,-179.777,8.294,149.528
C04323=1129.110,120.683,-57.580,-179.780,8.291,149.527
C04324=1129.116,120.434,-57.561,-179.782,8.287,149.527
C04325=1129.120,120.185,-57.541,-179.783,8.284,149.527
C04326=1129.125,119.936,-57.521,-179.785,8.281,149.527
C04327=1129.130,119.686,-57.501,-179.787,8.277,149.526
C04328=1129.135,119.437,-57.482,-179.789,8.274,149.526
C04329=1129.139,119.188,-57.462,-179.791,8.270,149.526
C04330=1129.144,118.939,-57.442,-179.792,8.267,149.525
C04331=1129.149,118.690,-57.423,-179.794,8.264,149.525
C04332=1129.154,118.441,-57.402,-179.796,8.260,149.525
C04333=1129.159,118.191,-57.383,-179.798,8.257,149.525
C04334=1129.163,117.942,-57.363,-179.800,8.253,149.525
C04335=1129.168,117.693,-57.344,-179.802,8.250,149.524
C04336=1129.172,117.478,-57.327,-179.804,8.247,149.524
C04337=1129.176,117.264,-57.311,-179.805,8.244,149.524
C04338=1129.180,117.049,-57.293,-179.807,8.240,149.523
C04339=1129.184,116.834,-57.276,-179.808,8.238,149.523
C04340=1129.189,116.620,-57.259,-179.810,8.235,149.523
C04341=1129.193,116.405,-57.242,-179.812,8.231,149.523
C04342=1129.197,116.190,-57.225,-179.813,8.229,149.523
C04343=1129.201,115.975,-57.208,-179.814,8.226,149.522
C04344=1129.206,115.725,-57.189,-179.817,8.223,149.522
C04345=1129.211,115.477,-57.169,-179.819,8.219,149.522
C04346=1129.215,115.227,-57.150,-179.821,8.216,149.522
C04347=1129.220,114.978,-57.131,-179.823,8.212,149.521
C04348=1129.225,114.729,-57.111,-179.824,8.208,149.521
C04349=1129.230,114.479,-57.092,-179.826,8.205,149.521
C04350=1129.234,114.230,-57.071,-179.828,8.201,149.521
C04351=1129.240,113.982,-57.052,-179.831,8.198,149.520
C04352=1129.244,113.732,-57.033,-179.833,8.194,149.520
C04353=1129.249,113.483,-57.014,-179.834,8.190,149.520
C04354=1129.254,113.234,-56.994,-179.836,8.187,149.520
C04355=1129.259,112.984,-56.974,-179.838,8.184,149.519
C04356=1129.263,112.736,-56.956,-179.840,8.181,149.519
C04357=1129.268,112.486,-56.936,-179.842,8.177,149.519
C04358=1129.273,112.237,-56.917,-179.843,8.173,149.518
C04359=1129.278,111.988,-56.897,-179.846,8.170,149.518
C04360=1129.282,111.738,-56.878,-179.848,8.166,149.518
C04361=1129.287,111.490,-56.859,-179.850,8.163,149.518
C04362=1129.292,111.240,-56.839,-179.852,8.159,149.518
C04363=1129.298,110.991,-56.820,-179.853,8.155,149.517
C04364=1129.302,110.741,-56.801,-179.856,8.151,149.517
C04365=1129.307,110.492,-56.782,-179.859,8.148,149.517
C04366=1129.312,110.243,-56.762,-179.861,8.144,149.517
C04367=1129.317,109.994,-56.744,-179.864,8.139,149.516
C04368=1129.321,109.745,-56.724,-179.866,8.136,149.516
C04369=1129.327,109.496,-56.705,-179.869,8.132,149.516
C04370=1129.331,109.247,-56.686,-179.871,8.127,149.516
C04371=1129.336,108.997,-56.667,-179.873,8.124,149.516
C04372=1129.340,108.748,-56.648,-179.877,8.120,149.516
C04373=1129.346,108.499,-56.629,-179.879,8.116,149.515
C04374=1129.350,108.249,-56.609,-179.881,8.112,149.515
C04375=1129.355,108.001,-56.590,-179.884,8.108,149.515
C04376=1129.360,107.751,-56.572,-179.886,8.104,149.515
C04377=1129.365,107.502,-56.553,-179.889,8.100,149.514
C04378=1129.369,107.253,-56.533,-179.891,8.096,149.514
C04379=1129.374,107.003,-56.515,-179.893,8.092,149.514
C04380=1129.379,106.754,-56.496,-179.896,8.088,149.514
C04381=1129.384,106.505,-56.477,-179.898,8.084,149.513
C04382=1129.389,106.255,-56.458,-179.900,8.080,149.513
C04383=1129.393,106.007,-56.439,-179.902,8.076,149.513
C04384=1129.398,105.757,-56.420,-179.905,8.072,149.513
C04385=1129.403,105.508,-56.402,-179.907,8.069,149.513
C04386=1129.408,105.259,-56.382,-179.909,8.064,149.512
C04387=1129.412,105.010,-56.363,-179.912,8.060,149.512
C04388=1129.418,104.760,-56.345,-179.914,8.056,149.512
C04389=1129.422,104.511,-56.326,-179.917,8.052,149.511
C04390=1129.428,104.261,-56.307,-179.919,8.048,149.511
C04391=1129.432,104.013,-56.288,-179.921,8.044,149.511
C04392=1129.436,103.797,-56.272,-179.923,8.041,149.511
C04393=1129.440,103.583,-56.256,-179.925,8.037,149.510
C04394=1129.445,103.368,-56.240,-179.927,8.034,149.510
C04395=1129.448,103.153,-56.223,-179.929,8.030,149.510
C04396=1129.453,102.938,-56.207,-179.931,8.027,149.510
C04397=1129.457,102.723,-56.192,-179.932,8.023,149.509
C04398=1129.461,102.508,-56.175,-179.934,8.020,149.509
C04399=1129.465,102.294,-56.160,-179.936,8.017,149.509
C04400=1129.470,102.044,-56.140,-179.939,8.013,149.509
C04401=1129.475,101.795,-56.122,-179.940,8.009,149.508
C04402=1129.480,101.546,-56.104,-179.942,8.005,149.508
C04403=1129.485,101.296,-56.084,-179.945,8.000,149.508
C04404=1129.490,101.047,-56.066,-179.947,7.997,149.507
C04405=1129.494,100.798,-56.048,-179.949,7.992,149.507
C04406=1129.500,100.549,-56.029,-179.951,7.989,149.507
C04407=1129.504,100.299,-56.011,-179.952,7.985,149.506
C04408=1129.509,100.050,-55.992,-179.955,7.981,149.506
C04409=1129.515,99.801,-55.973,-179.957,7.977,149.506
C04410=1129.519,99.551,-55.955,-179.958,7.973,149.505
C04411=1129.524,99.302,-55.937,-179.961,7.969,149.505
C04412=1129.528,99.053,-55.918,-179.963,7.965,149.505
C04413=1129.534,98.804,-55.900,-179.965,7.961,149.504
C04414=1129.538,98.554,-55.882,-179.967,7.956,149.504
C04415=1129.543,98.305,-55.863,-179.969,7.953,149.503
C04416=1129.548,98.056,-55.845,-179.971,7.949,149.503
C04417=1129.553,97.807,-55.826,-179.973,7.944,149.503
C04418=1129.558,97.557,-55.808,-179.974,7.941,149.502
C04419=1129.563,97.308,-55.790,-179.976,7.937,149.502
C04420=1129.567,97.059,-55.771,-179.978,7.933,149.502
C04421=1129.572,96.810,-55.753,-179.980,7.928,149.501
C04422=1129.577,96.560,-55.734,-179.982,7.925,149.501
C04423=1129.582,96.311,-55.716,-179.984,7.921,149.501
C04424=1129.587,96.061,-55.698,-179.986,7.917,149.500
C04425=1129.592,95.812,-55.680,-179.987,7.913,149.500
C04426=1129.597,95.563,-55.662,-179.989,7.909,149.499
C04427=1129.601,95.313,-55.644,-179.991,7.905,149.499
C04428=1129.606,95.065,-55.625,-179.993,7.901,149.499
C04429=1129.611,94.815,-55.607,-179.995,7.897,149.498
C04430=1129.616,94.566,-55.589,-179.996,7.893,149.498
C04431=1129.621,94.317,-55.571,-179.998,7.890,149.498
C04432=1129.626,94.068,-55.553,180.000,7.885,149.497
C04433=1129.631,93.818,-55.535,179.998,7.881,149.497
C04434=1129.635,93.569,-55.517,179.997,7.877,149.496
C04435=1129.640,93.319,-55.499,179.995,7.873,149.496
C04436=1129.645,93.070,-55.481,179.994,7.869,149.495
C04437=1129.650,92.821,-55.463,179.992,7.865,149.495
C04438=1129.655,92.572,-55.445,179.990,7.862,149.495
C04439=1129.660,92.323,-55.427,179.989,7.858,149.494
C04440=1129.665,92.074,-55.409,179.987,7.854,149.494
C04441=1129.670,91.823,-55.391,179.986,7.850,149.493
C04442=1129.674,91.574,-55.373,179.984,7.846,149.493
C04443=1129.679,91.325,-55.355,179.982,7.842,149.492
C04444=1129.684,91.075,-55.337,179.981,7.838,149.492
C04445=1129.689,90.826,-55.319,179.979,7.834,149.492
C04446=1129.694,90.577,-55.301,179.977,7.830,149.491
C04447=1129.699,90.328,-55.283,179.975,7.826,149.491
C04448=1129.703,90.113,-55.268,179.974,7.823,149.490
C04449=1129.708,89.898,-55.252,179.973,7.820,149.490
C04450=1129.712,89.682,-55.237,179.972,7.816,149.489
C04451=1129.716,89.467,-55.221,179.970,7.813,149.489
C04452=1129.720,89.253,-55.206,179.969,7.809,149.489
C04453=1129.724,89.038,-55.191,179.968,7.806,149.488
C04454=1129.729,88.823,-55.176,179.967,7.803,149.488
C04455=1129.733,88.608,-55.161,179.965,7.799,149.487
C04456=1129.738,88.359,-55.143,179.964,7.795,149.487
C04457=1129.743,88.110,-55.125,179.962,7.791,149.487
C04458=1129.748,87.860,-55.107,179.960,7.787,149.486
C04459=1129.753,87.611,-55.089,179.960,7.784,149.486
C04460=1129.758,87.361,-55.071,179.958,7.780,149.485
C04461=1129.763,87.112,-55.053,179.957,7.776,149.485
C04462=1129.768,86.862,-55.036,179.955,7.772,149.484
C04463=1129.772,86.614,-55.019,179.954,7.768,149.484
C04464=1129.777,86.364,-55.001,179.952,7.764,149.483
C04465=1129.782,86.115,-54.983,179.951,7.760,149.483
C04466=1129.787,85.865,-54.965,179.950,7.757,149.482
C04467=1129.792,85.616,-54.948,179.949,7.753,149.482
C04468=1129.797,85.366,-54.930,179.947,7.749,149.481
C04469=1129.801,85.118,-54.913,179.946,7.745,149.481
C04470=1129.806,84.868,-54.895,179.945,7.741,149.480
C04471=1129.811,84.619,-54.878,179.943,7.737,149.480
C04472=1129.816,84.369,-54.860,179.942,7.733,149.479
C04473=1129.822,84.120,-54.842,179.941,7.729,149.479
C04474=1129.826,83.871,-54.825,179.940,7.726,149.478
C04475=1129.831,83.622,-54.807,179.938,7.722,149.478
C04476=1129.836,83.372,-54.790,179.937,7.718,149.477
C04477=1129.841,83.123,-54.772,179.935,7.714,149.477
C04478=1129.845,82.873,-54.755,179.935,7.710,149.476
C04479=1129.850,82.624,-54.737,179.933,7.707,149.476
C04480=1129.855,82.374,-54.720,179.932,7.703,149.475
C04481=1129.860,82.125,-54.702,179.931,7.699,149.475
C04482=1129.865,81.875,-54.685,179.930,7.695,149.474
C04483=1129.870,81.626,-54.667,179.929,7.691,149.474
C04484=1129.875,81.376,-54.650,179.928,7.688,149.473
C04485=1129.880,81.128,-54.632,179.926,7.684,149.473
C04486=1129.885,80.879,-54.616,179.926,7.681,149.472
C04487=1129.890,80.629,-54.598,179.924,7.676,149.471
C04488=1129.895,80.380,-54.580,179.923,7.672,149.471
C04489=1129.899,80.131,-54.563,179.922,7.669,149.470
C04490=1129.904,79.881,-54.546,179.921,7.665,149.470
C04491=1129.910,79.631,-54.529,179.920,7.661,149.469
C04492=1129.914,79.382,-54.511,179.919,7.658,149.469
C04493=1129.920,79.133,-54.494,179.918,7.654,149.468
C04494=1129.925,78.884,-54.476,179.917,7.650,149.468
C04495=1129.929,78.635,-54.460,179.916,7.647,149.467
C04496=1129.934,78.385,-54.442,179.914,7.643,149.467
C04497=1129.939,78.136,-54.424,179.914,7.639,149.466
C04498=1129.944,77.886,-54.408,179.912,7.635,149.466
C04499=1129.949,77.636,-54.390,179.912,7.632,149.465
C04500=1129.954,77.388,-54.373,179.911,7.628,149.464
C04501=1129.959,77.138,-54.356,179.910,7.624,149.464
C04502=1129.964,76.888,-54.339,179.909,7.621,149.463
C04503=1129.968,76.640,-54.321,179.908,7.617,149.463
C04504=1129.973,76.424,-54.307,179.907,7.614,149.462
C04505=1129.977,76.209,-54.292,179.905,7.610,149.462
C04506=1129.981,75.994,-54.277,179.904,7.607,149.462
C04507=1129.986,75.779,-54.262,179.903,7.603,149.461
C04508=1129.989,75.564,-54.248,179.902,7.600,149.461
C04509=1129.994,75.348,-54.233,179.901,7.597,149.460
C04510=1129.998,75.134,-54.218,179.899,7.593,149.460
C04511=1130.002,74.918,-54.203,179.898,7.590,149.460
C04512=1130.007,74.670,-54.187,179.897,7.586,149.459
C04513=1130.013,74.420,-54.170,179.895,7.582,149.459
C04514=1130.017,74.171,-54.152,179.893,7.578,149.458
C04515=1130.022,73.921,-54.135,179.892,7.574,149.458
C04516=1130.027,73.672,-54.118,179.891,7.570,149.457
C04517=1130.032,73.423,-54.102,179.889,7.566,149.457
C04518=1130.037,73.173,-54.085,179.888,7.562,149.456
C04519=1130.042,72.923,-54.068,179.886,7.558,149.456
C04520=1130.047,72.674,-54.051,179.885,7.554,149.455
C04521=1130.052,72.425,-54.033,179.883,7.550,149.455
C04522=1130.057,72.176,-54.017,179.882,7.546,149.454
C04523=1130.062,71.926,-53.999,179.881,7.542,149.454
C04524=1130.066,71.677,-53.983,179.879,7.538,149.453
C04525=1130.072,71.427,-53.966,179.877,7.534,149.453
C04526=1130.077,71.178,-53.949,179.876,7.530,149.452
C04527=1130.081,70.929,-53.932,179.875,7.526,149.452
C04528=1130.087,70.679,-53.916,179.873,7.522,149.451
C04529=1130.091,70.430,-53.899,179.872,7.518,149.451
C04530=1130.097,70.180,-53.882,179.870,7.514,149.451
C04531=1130.102,69.931,-53.865,179.869,7.510,149.450
C04532=1130.106,69.682,-53.849,179.867,7.506,149.449
C04533=1130.111,69.432,-53.831,179.866,7.502,149.449
C04534=1130.116,69.183,-53.815,179.864,7.498,149.449
C04535=1130.121,68.934,-53.798,179.863,7.494,149.448
C04536=1130.126,68.684,-53.781,179.861,7.490,149.448
C04537=1130.131,68.435,-53.764,179.860,7.486,149.447
C04538=1130.136,68.186,-53.748,179.859,7.482,149.447
C04539=1130.141,67.936,-53.731,179.857,7.478,149.446
C04540=1130.146,67.687,-53.715,179.856,7.474,149.446
C04541=1130.150,67.438,-53.698,179.854,7.470,149.445
C04542=1130.156,67.187,-53.681,179.853,7.466,149.445
C04543=1130.161,66.938,-53.665,179.851,7.462,149.444
C04544=1130.165,66.689,-53.648,179.850,7.458,149.444
C04545=1130.170,66.440,-53.632,179.849,7.454,149.443
C04546=1130.176,66.190,-53.615,179.847,7.450,149.443
C04547=1130.180,65.941,-53.598,179.846,7.446,149.442
C04548=1130.185,65.691,-53.582,179.844,7.442,149.442
C04549=1130.190,65.442,-53.566,179.843,7.438,149.441
C04550=1130.195,65.192,-53.549,179.841,7.434,149.441
C04551=1130.200,64.943,-53.532,179.840,7.430,149.440
C04552=1130.205,64.694,-53.516,179.839,7.425,149.440
C04553=1130.210,64.444,-53.500,179.837,7.421,149.439
C04554=1130.216,64.195,-53.483,179.836,7.418,149.439
C04555=1130.220,63.945,-53.466,179.834,7.413,149.438
C04556=1130.225,63.697,-53.450,179.833,7.409,149.438
C04557=1130.230,63.446,-53.434,179.831,7.405,149.437
C04558=1130.235,63.198,-53.418,179.831,7.402,149.437
C04559=1130.239,62.948,-53.401,179.829,7.398,149.436
C04560=1130.248,62.532,-53.373,179.827,7.391,149.435
C04561=1130.257,62.116,-53.347,179.824,7.384,149.435
C04562=1130.265,61.699,-53.319,179.822,7.378,149.434
C04563=1130.273,61.283,-53.292,179.819,7.371,149.433
C04564=1130.278,61.034,-53.275,179.818,7.367,149.432
C04565=1130.283,60.784,-53.259,179.817,7.363,149.432
C04566=1130.288,60.535,-53.243,179.815,7.359,149.432
C04567=1130.293,60.285,-53.227,179.814,7.355,149.431
C04568=1130.298,60.036,-53.211,179.812,7.351,149.431
C04569=1130.303,59.787,-53.194,179.811,7.346,149.430
C04570=1130.308,59.538,-53.178,179.810,7.343,149.429
C04571=1130.313,59.288,-53.162,179.808,7.339,149.429
C04572=1130.318,59.039,-53.146,179.807,7.334,149.428
C04573=1130.322,58.789,-53.129,179.806,7.330,149.428
C04574=1130.328,58.540,-53.114,179.804,7.327,149.428
C04575=1130.332,58.290,-53.097,179.803,7.322,149.427
C04576=1130.338,58.041,-53.082,179.801,7.318,149.426
C04577=1130.342,57.791,-53.065,179.800,7.314,149.426
C04578=1130.348,57.542,-53.049,179.799,7.310,149.425
C04579=1130.352,57.292,-53.033,179.797,7.306,149.425
C04580=1130.357,57.043,-53.017,179.796,7.302,149.424
C04581=1130.363,56.794,-53.001,179.794,7.298,149.424
C04582=1130.367,56.544,-52.985,179.793,7.294,149.423
C04583=1130.373,56.295,-52.969,179.792,7.290,149.423
C04584=1130.377,56.045,-52.953,179.790,7.286,149.422
C04585=1130.383,55.796,-52.937,179.789,7.282,149.422
C04586=1130.388,55.547,-52.921,179.788,7.278,149.421
C04587=1130.392,55.297,-52.905,179.786,7.273,149.421
C04588=1130.398,55.048,-52.889,179.785,7.269,149.420
C04589=1130.403,54.798,-52.873,179.783,7.266,149.420
C04590=1130.408,54.549,-52.857,179.782,7.261,149.419
C04591=1130.413,54.299,-52.841,179.781,7.257,149.419
C04592=1130.418,54.049,-52.825,179.780,7.253,149.418
C04593=1130.423,53.800,-52.809,179.778,7.249,149.418
C04594=1130.428,53.551,-52.793,179.777,7.245,149.417
C04595=1130.432,53.301,-52.778,179.775,7.241,149.417
C04596=1130.438,53.052,-52.763,179.774,7.237,149.416
C04597=1130.442,52.802,-52.746,179.773,7.233,149.416
C04598=1130.448,52.553,-52.730,179.771,7.229,149.415
C04599=1130.453,52.304,-52.715,179.770,7.224,149.415
C04600=1130.458,52.053,-52.699,179.769,7.221,149.414
C04601=1130.463,51.805,-52.682,179.767,7.216,149.413
C04602=1130.467,51.556,-52.667,179.766,7.212,149.413
C04603=1130.473,51.306,-52.652,179.765,7.208,149.412
C04604=1130.478,51.056,-52.636,179.763,7.204,149.412
C04605=1130.483,50.807,-52.620,179.762,7.200,149.411
C04606=1130.488,50.557,-52.605,179.761,7.196,149.411
C04607=1130.492,50.308,-52.589,179.760,7.192,149.410
C04608=1130.518,49.073,-52.511,-179.936,6.565,149.182
C04609=1130.526,48.662,-52.485,-179.940,6.562,149.183
C04610=1130.531,48.413,-52.470,-179.943,6.561,149.183
C04611=1130.536,48.163,-52.455,-179.946,6.560,149.184
C04612=1130.541,47.913,-52.439,-179.948,6.559,149.184
C04613=1130.546,47.664,-52.424,-179.951,6.557,149.185
C04614=1130.551,47.415,-52.409,-179.953,6.557,149.185
C04615=1130.556,47.166,-52.394,-179.956,6.555,149.186
C04616=1130.561,46.916,-52.378,-179.959,6.553,149.186
C04617=1130.566,46.666,-52.362,-179.961,6.553,149.187
C04618=1130.571,46.417,-52.347,-179.964,6.551,149.187
C04619=1130.576,46.168,-52.332,-179.966,6.551,149.188
C04620=1130.581,45.918,-52.317,-179.969,6.549,149.188
C04621=1130.586,45.669,-52.302,-179.972,6.548,149.189
C04622=1130.592,45.419,-52.286,-179.974,6.547,149.189
C04623=1130.596,45.169,-52.271,-179.977,6.545,149.190
C04624=1130.601,44.920,-52.255,-179.979,6.544,149.190
C04625=1130.606,44.670,-52.241,-179.983,6.543,149.191
C04626=1130.611,44.421,-52.225,-179.985,6.542,149.191
C04627=1130.616,44.172,-52.210,-179.988,6.541,149.192
C04628=1130.621,43.922,-52.195,-179.990,6.540,149.193
C04629=1130.626,43.673,-52.180,-179.993,6.539,149.193
C04630=1130.632,43.423,-52.165,-179.996,6.537,149.193
C04631=1130.636,43.173,-52.150,-179.998,6.536,149.194
C04632=1130.641,42.924,-52.134,179.999,6.535,149.195
C04633=1130.646,42.675,-52.119,179.997,6.534,149.195
C04634=1130.652,42.425,-52.104,179.994,6.532,149.196
C04635=1130.656,42.176,-52.089,179.992,6.532,149.196
C04636=1130.662,41.926,-52.074,179.989,6.530,149.197
C04637=1130.667,41.677,-52.059,179.986,6.530,149.197
C04638=1130.672,41.427,-52.044,179.984,6.528,149.198
C04639=1130.677,41.178,-52.029,179.981,6.528,149.198
C04640=1130.682,40.928,-52.014,179.978,6.526,149.199
C04641=1130.687,40.679,-51.999,179.975,6.524,149.199
C04642=1130.692,40.430,-51.983,179.973,6.523,149.200
C04643=1130.697,40.179,-51.969,179.970,6.522,149.200
C04644=1130.702,39.930,-51.953,179.968,6.521,149.201
C04645=1130.707,39.680,-51.939,179.965,6.520,149.201
C04646=1130.712,39.431,-51.924,179.962,6.519,149.202
C04647=1130.717,39.182,-51.908,179.960,6.518,149.202
C04648=1130.722,38.932,-51.894,179.958,6.517,149.203
C04649=1130.727,38.683,-51.878,179.955,6.515,149.203
C04650=1130.732,38.433,-51.864,179.952,6.515,149.204
C04651=1130.737,38.184,-51.849,179.949,6.513,149.204
C04652=1130.743,37.934,-51.834,179.947,6.512,149.205
C04653=1130.747,37.685,-51.819,179.944,6.511,149.205
C04654=1130.752,37.435,-51.805,179.942,6.510,149.206
C04655=1130.758,37.186,-51.789,179.939,6.509,149.206
C04656=1130.763,36.936,-51.775,179.937,6.508,149.207
C04657=1130.767,36.687,-51.760,179.934,6.507,149.207
C04658=1130.773,36.437,-51.745,179.931,6.506,149.208
C04659=1130.778,36.188,-51.730,179.929,6.504,149.208
C04660=1130.783,35.938,-51.716,179.926,6.504,149.209
C04661=1130.788,35.689,-51.700,179.923,6.502,149.209
C04662=1130.793,35.439,-51.686,179.921,6.501,149.210
C04663=1130.798,35.190,-51.671,179.918,6.500,149.210
C04664=1130.803,34.940,-51.656,179.916,6.499,149.211
C04665=1130.809,34.691,-51.642,179.913,6.498,149.211
C04666=1130.813,34.442,-51.627,179.911,6.497,149.212
C04667=1130.819,34.192,-51.612,179.907,6.496,149.213
C04668=1130.824,33.943,-51.597,179.905,6.495,149.213
C04669=1130.829,33.693,-51.583,179.903,6.493,149.214
C04670=1130.834,33.443,-51.569,179.900,6.492,149.214
C04671=1130.839,33.194,-51.553,179.897,6.491,149.215
C04672=1130.844,32.944,-51.539,179.895,6.490,149.215
C04673=1130.849,32.694,-51.525,179.892,6.489,149.216
C04674=1130.854,32.445,-51.510,179.890,6.488,149.216
C04675=1130.859,32.195,-51.495,179.887,6.487,149.217
C04676=1130.864,31.945,-51.481,179.885,6.486,149.217
C04677=1130.869,31.696,-51.466,179.882,6.484,149.218
C04678=1130.874,31.447,-51.451,179.879,6.484,149.218
C04679=1130.879,31.198,-51.437,179.876,6.482,149.219
C04680=1130.884,30.948,-51.423,179.874,6.481,149.219
C04681=1130.890,30.699,-51.408,179.871,6.480,149.220
C04682=1130.895,30.449,-51.393,179.869,6.479,149.220
C04683=1130.900,30.199,-51.379,179.867,6.478,149.221
C04684=1130.905,29.949,-51.365,179.863,6.477,149.221
C04685=1130.909,29.700,-51.350,179.861,6.476,149.222
C04686=1130.914,29.451,-51.335,179.858,6.475,149.222
C04687=1130.921,29.201,-51.321,179.856,6.474,149.223
C04688=1130.926,28.952,-51.307,179.853,6.473,149.223
C04689=1130.930,28.702,-51.292,179.851,6.472,149.224
C04690=1130.935,28.453,-51.277,179.848,6.470,149.224
C04691=1130.940,28.203,-51.263,179.845,6.470,149.225
C04692=1130.945,27.953,-51.249,179.843,6.468,149.226
C04693=1130.950,27.704,-51.235,179.841,6.467,149.226
C04694=1130.956,27.436,-51.219,179.837,6.466,149.227
C04695=1130.962,27.166,-51.204,179.835,6.465,149.227
C04696=1130.967,26.897,-51.188,179.832,6.464,149.228
C04697=1130.972,26.628,-51.173,179.829,6.463,149.228
C04698=1130.977,26.378,-51.159,179.827,6.462,149.229
C04699=1130.982,26.129,-51.144,179.824,6.461,149.229
C04700=1130.988,25.880,-51.130,179.821,6.460,149.230
C04701=1130.993,25.630,-51.115,179.819,6.459,149.230
C04702=1130.998,25.380,-51.101,179.816,6.458,149.231
C04703=1131.002,25.131,-51.087,179.814,6.457,149.231
C04704=1131.007,24.881,-51.073,179.811,6.455,149.232
C04705=1131.013,24.632,-51.059,179.808,6.455,149.233
C04706=1131.018,24.382,-51.044,179.806,6.454,149.233
C04707=1131.023,24.133,-51.030,179.804,6.452,149.233
C04708=1131.028,23.883,-51.016,179.801,6.452,149.234
C04709=1131.033,23.634,-51.002,179.798,6.450,149.235
C04710=1131.038,23.384,-50.988,179.796,6.449,149.235
C04711=1131.043,23.134,-50.973,179.794,6.449,149.236
C04712=1131.048,22.885,-50.959,179.791,6.447,149.236
C04713=1131.054,22.636,-50.945,179.788,6.447,149.237
C04714=1131.059,22.386,-50.931,179.786,6.445,149.237
C04715=1131.064,22.136,-50.917,179.783,6.445,149.238
C04716=1131.069,21.887,-50.902,179.781,6.444,149.238
C04717=1131.074,21.638,-50.889,179.778,6.442,149.239
C04718=1131.080,21.387,-50.875,179.775,6.442,149.239
C04719=1131.084,21.137,-50.861,179.773,6.440,149.240
C04720=1131.089,20.888,-50.846,179.770,6.439,149.240
C04721=1131.095,20.639,-50.832,179.768,6.439,149.241
C04722=1131.100,20.389,-50.818,179.765,6.437,149.241
C04723=1131.105,20.139,-50.804,179.763,6.436,149.242
C04724=1131.110,19.890,-50.790,179.760,6.435,149.242
C04725=1131.115,19.641,-50.776,179.757,6.434,149.243
C04726=1131.120,19.391,-50.763,179.755,6.434,149.244
C04727=1131.125,19.142,-50.749,179.752,6.432,149.244
C04728=1131.130,18.892,-50.735,179.750,6.432,149.245
C04729=1131.135,18.642,-50.720,179.747,6.430,149.245
C04730=1131.141,18.393,-50.706,179.745,6.429,149.246
C04731=1131.146,18.143,-50.693,179.742,6.429,149.246
C04732=1131.150,17.893,-50.679,179.739,6.427,149.247
C04733=1131.156,17.644,-50.665,179.737,6.426,149.247
C04734=1131.161,17.395,-50.651,179.735,6.426,149.248
C04735=1131.166,17.145,-50.637,179.732,6.424,149.248
C04736=1131.172,16.895,-50.623,179.730,6.423,149.249
C04737=1131.177,16.646,-50.609,179.727,6.423,149.249
C04738=1131.181,16.396,-50.596,179.724,6.421,149.250
C04739=1131.187,16.147,-50.582,179.722,6.421,149.250
C04740=1131.192,15.897,-50.568,179.719,6.419,149.251
C04741=1131.197,15.647,-50.554,179.717,6.419,149.252
C04742=1131.202,15.398,-50.540,179.714,6.418,149.252
C04743=1131.207,15.148,-50.527,179.712,6.416,149.252
C04744=1131.212,14.899,-50.513,179.709,6.416,149.253
C04745=1131.217,14.649,-50.499,179.707,6.415,149.254
C04746=1131.223,14.399,-50.485,179.704,6.413,149.254
C04747=1131.227,14.150,-50.472,179.701,6.413,149.255
C04748=1131.232,13.901,-50.458,179.699,6.412,149.255
C04749=1131.238,13.651,-50.444,179.696,6.410,149.256
C04750=1131.243,13.401,-50.430,179.694,6.410,149.256
C04751=1131.248,13.151,-50.417,179.692,6.409,149.257
C04752=1131.253,12.902,-50.403,179.689,6.408,149.257
C04753=1131.258,12.653,-50.389,179.687,6.407,149.258
C04754=1131.263,12.403,-50.376,179.684,6.406,149.258
C04755=1131.268,12.154,-50.362,179.681,6.405,149.259
C04756=1131.274,11.904,-50.349,179.679,6.404,149.259
C04757=1131.279,11.654,-50.335,179.676,6.404,149.260
C04758=1131.284,11.404,-50.322,179.674,6.402,149.260
C04759=1131.289,11.155,-50.308,179.671,6.401,149.261
C04760=1131.294,10.906,-50.293,179.669,6.401,149.262
C04761=1131.299,10.656,-50.281,179.666,6.399,149.262
C04762=1131.304,10.406,-50.267,179.664,6.398,149.263
C04763=1131.310,10.157,-50.253,179.661,6.398,149.263
C04764=1131.314,9.907,-50.240,179.658,6.396,149.264
C04765=1131.320,9.658,-50.226,179.656,6.396,149.264
C04766=1131.324,9.408,-50.213,179.654,6.395,149.265
C04767=1131.330,9.159,-50.200,179.651,6.394,149.265
C04768=1131.335,8.908,-50.186,179.649,6.393,149.266
C04769=1131.340,8.660,-50.173,179.646,6.392,149.266
C04770=1131.346,8.409,-50.159,179.643,6.391,149.267
C04771=1131.350,8.161,-50.146,179.641,6.390,149.267
C04772=1131.356,7.910,-50.132,179.639,6.389,149.268
C04773=1131.361,7.661,-50.118,179.636,6.389,149.269
C04774=1131.366,7.411,-50.105,179.633,6.387,149.269
C04775=1131.372,7.162,-50.092,179.631,6.386,149.269
C04776=1131.376,6.912,-50.079,179.629,6.386,149.270
C04777=1131.382,6.663,-50.065,179.626,6.384,149.271
C04778=1131.386,6.413,-50.052,179.624,6.383,149.271
C04779=1131.392,6.164,-50.038,179.621,6.383,149.272
C04780=1131.397,5.913,-50.025,179.618,6.381,149.272
C04781=1131.402,5.665,-50.012,179.616,6.381,149.273
C04782=1131.408,5.415,-49.998,179.613,6.380,149.273
C04783=1131.412,5.165,-49.985,179.611,6.379,149.274
C04784=1131.418,4.916,-49.971,179.608,6.378,149.274
C04785=1131.422,4.666,-49.959,179.606,6.377,149.275
C04786=1131.428,4.416,-49.945,179.604,6.377,149.275
C04787=1131.433,4.166,-49.932,179.601,6.375,149.276
C04788=1131.438,3.917,-49.918,179.598,6.375,149.277
C04789=1131.443,3.667,-49.905,179.596,6.374,149.277
C04790=1131.449,3.418,-49.892,179.594,6.373,149.278
C04791=1131.453,3.169,-49.879,179.591,6.371,149.278
C04792=1131.459,2.919,-49.865,179.588,6.371,149.279
C04793=1131.464,2.669,-49.853,179.586,6.370,149.279
C04794=1131.468,2.419,-49.840,179.584,6.369,149.280
C04795=1131.474,2.170,-49.827,179.581,6.368,149.280
C04796=1131.479,1.921,-49.813,179.579,6.367,149.281
C04797=1131.484,1.671,-49.800,179.576,6.367,149.281
C04798=1131.489,1.401,-49.786,179.573,6.365,149.282
C04799=1131.495,1.132,-49.771,179.571,6.365,149.282
C04800=1131.501,0.862,-49.757,179.568,6.363,149.283
C04801=1131.506,0.592,-49.744,179.566,6.363,149.284
C04802=1131.512,0.343,-49.730,179.563,6.362,149.284
C04803=1131.517,0.094,-49.718,179.561,6.361,149.285
C04804=1131.522,-0.156,-49.703,179.558,6.360,149.285
C04805=1131.527,-0.405,-49.691,179.555,6.359,149.286
C04806=1131.532,-0.655,-49.678,179.553,6.358,149.286
C04807=1131.537,-0.905,-49.665,179.551,6.358,149.287
C04808=1131.543,-1.154,-49.652,179.548,6.356,149.288
C04809=1131.548,-1.404,-49.639,179.545,6.356,149.288
C04810=1131.553,-1.654,-49.626,179.543,6.355,149.288
C04811=1131.558,-1.903,-49.613,179.541,6.354,149.289
C04812=1131.563,-2.153,-49.601,179.538,6.353,149.290
C04813=1131.568,-2.403,-49.587,179.536,6.352,149.290
C04814=1131.574,-2.652,-49.575,179.534,6.351,149.291
C04815=1131.578,-2.901,-49.561,179.531,6.351,149.291
C04816=1131.584,-3.151,-49.548,179.528,6.349,149.292
C04817=1131.589,-3.401,-49.535,179.526,6.348,149.292
C04818=1131.594,-3.650,-49.522,179.523,6.348,149.293
C04819=1131.599,-3.900,-49.509,179.521,6.347,149.293
C04820=1131.604,-4.150,-49.496,179.519,6.346,149.294
C04821=1131.609,-4.399,-49.484,179.516,6.345,149.294
C04822=1131.615,-4.649,-49.471,179.513,6.344,149.295
C04823=1131.620,-4.899,-49.458,179.511,6.344,149.295
C04824=1131.625,-5.148,-49.445,179.509,6.343,149.296
C04825=1131.630,-5.398,-49.433,179.506,6.342,149.297
C04826=1131.636,-5.648,-49.420,179.504,6.341,149.297
C04827=1131.641,-5.898,-49.407,179.501,6.340,149.298
C04828=1131.646,-6.147,-49.394,179.499,6.340,149.298
C04829=1131.651,-6.396,-49.382,179.497,6.339,149.299
C04830=1131.656,-6.647,-49.368,179.494,6.337,149.299
C04831=1131.661,-6.896,-49.356,179.491,6.337,149.300
C04832=1131.667,-7.145,-49.343,179.489,6.336,149.300
C04833=1131.672,-7.394,-49.330,179.487,6.335,149.301
C04834=1131.677,-7.644,-49.318,179.484,6.335,149.301
C04835=1131.682,-7.894,-49.304,179.481,6.333,149.302
C04836=1131.687,-8.144,-49.292,179.479,6.332,149.302
C04837=1131.693,-8.393,-49.280,179.477,6.332,149.303
C04838=1131.698,-8.643,-49.267,179.474,6.331,149.304
C04839=1131.702,-8.893,-49.254,179.472,6.330,149.304
C04840=1131.708,-9.142,-49.241,179.469,6.329,149.305
C04841=1131.713,-9.392,-49.228,179.467,6.328,149.305
C04842=1131.719,-9.642,-49.216,179.465,6.328,149.306
C04843=1131.724,-9.891,-49.204,179.462,6.327,149.306
C04844=1131.728,-10.141,-49.191,179.460,6.326,149.307
C04845=1131.733,-10.390,-49.178,179.458,6.326,149.307
C04846=1131.739,-10.640,-49.166,179.454,6.325,149.308
C04847=1131.745,-10.890,-49.153,179.452,6.324,149.308
C04848=1131.750,-11.139,-49.141,179.450,6.323,149.309
C04849=1131.754,-11.389,-49.128,179.448,6.322,149.309
C04850=1131.759,-11.638,-49.115,179.445,6.322,149.310
C04851=1131.765,-11.888,-49.103,179.443,6.321,149.311
C04852=1131.770,-12.138,-49.091,179.440,6.319,149.311
C04853=1131.775,-12.387,-49.078,179.437,6.319,149.312
C04854=1131.780,-12.636,-49.065,179.435,6.318,149.312
C04855=1131.785,-12.887,-49.053,179.433,6.317,149.313
C04856=1131.790,-13.136,-49.040,179.430,6.317,149.313
C04857=1131.795,-13.386,-49.028,179.428,6.316,149.314
C04858=1131.802,-13.636,-49.015,179.425,6.315,149.314
C04859=1131.807,-13.885,-49.003,179.423,6.314,149.315
C04860=1131.812,-14.135,-48.990,179.421,6.313,149.315
C04861=1131.817,-14.384,-48.978,179.418,6.313,149.316
C04862=1131.822,-14.634,-48.965,179.416,6.312,149.316
C04863=1131.827,-14.884,-48.953,179.414,6.311,149.317
C04864=1131.832,-15.134,-48.941,179.411,6.310,149.318
C04865=1131.837,-15.383,-48.928,179.409,6.309,149.318
C04866=1131.843,-15.633,-48.916,179.406,6.309,149.319
C04867=1131.848,-15.882,-48.904,179.404,6.308,149.319
C04868=1131.853,-16.132,-48.891,179.402,6.307,149.320
C04869=1131.858,-16.382,-48.879,179.399,6.307,149.320
C04870=1131.864,-16.631,-48.867,179.397,6.306,149.321
C04871=1131.869,-16.881,-48.855,179.395,6.305,149.321
C04872=1131.874,-17.131,-48.842,179.391,6.304,149.322
C04873=1131.879,-17.381,-48.830,179.389,6.303,149.322
C04874=1131.884,-17.630,-48.817,179.387,6.302,149.323
C04875=1131.889,-17.879,-48.805,179.385,6.301,149.323
C04876=1131.895,-18.129,-48.793,179.382,6.301,149.324
C04877=1131.900,-18.379,-48.780,179.380,6.300,149.325
C04878=1131.905,-18.629,-48.768,179.378,6.299,149.325
C04879=1131.910,-18.878,-48.756,179.374,6.298,149.326
C04880=1131.915,-19.128,-48.744,179.372,6.298,149.326
C04881=1131.920,-19.377,-48.732,179.370,6.297,149.327
C04882=1131.926,-19.627,-48.720,179.367,6.296,149.327
C04883=1131.931,-19.876,-48.707,179.365,6.296,149.328
C04884=1131.936,-20.126,-48.696,179.363,6.295,149.328
C04885=1131.942,-20.376,-48.684,179.361,6.294,149.329
C04886=1131.947,-20.625,-48.671,179.358,6.294,149.329
C04887=1131.952,-20.875,-48.659,179.356,6.293,149.330
C04888=1131.957,-21.125,-48.647,179.353,6.291,149.330
C04889=1131.963,-21.374,-48.635,179.351,6.291,149.331
C04890=1131.968,-21.624,-48.622,179.348,6.290,149.332
C04891=1131.973,-21.873,-48.611,179.346,6.289,149.332
C04892=1131.978,-22.123,-48.599,179.344,6.289,149.333
C04893=1131.983,-22.373,-48.586,179.341,6.288,149.333
C04894=1131.988,-22.623,-48.574,179.339,6.287,149.334
C04895=1131.994,-22.873,-48.563,179.337,6.287,149.334
C04896=1131.999,-23.122,-48.550,179.334,6.286,149.335
C04897=1132.004,-23.372,-48.538,179.332,6.285,149.335
C04898=1132.009,-23.621,-48.526,179.329,6.284,149.336
C04899=1132.014,-23.871,-48.514,179.327,6.283,149.337
C04900=1132.020,-24.121,-48.502,179.325,6.283,149.337
C04901=1132.025,-24.371,-48.490,179.322,6.282,149.337
C04902=1132.030,-24.640,-48.477,179.320,6.281,149.338
C04903=1132.036,-24.910,-48.464,179.317,6.281,149.339
C04904=1132.041,-25.180,-48.451,179.314,6.279,149.339
C04905=1132.047,-25.451,-48.438,179.312,6.279,149.340
C04906=1132.052,-25.701,-48.426,179.309,6.278,149.340
C04907=1132.058,-25.951,-48.414,179.307,6.277,149.341
C04908=1132.064,-26.200,-48.403,179.305,6.277,149.341
C04909=1132.069,-26.449,-48.390,179.303,6.276,149.342
C04910=1132.073,-26.699,-48.379,179.300,6.275,149.343
C04911=1132.079,-26.949,-48.367,179.298,6.275,149.343
C04912=1132.084,-27.199,-48.355,179.296,6.274,149.344
C04913=1132.089,-27.448,-48.343,179.293,6.273,149.344
C04914=1132.094,-27.698,-48.331,179.291,6.273,149.345
C04915=1132.099,-27.948,-48.319,179.288,6.271,149.345
C04916=1132.105,-28.197,-48.308,179.286,6.270,149.346
C04917=1132.110,-28.447,-48.296,179.283,6.270,149.346
C04918=1132.115,-28.696,-48.284,179.281,6.269,149.347
C04919=1132.120,-28.946,-48.272,179.279,6.268,149.347
C04920=1132.126,-29.196,-48.260,179.276,6.268,149.348
C04921=1132.131,-29.445,-48.249,179.274,6.267,149.348
C04922=1132.136,-29.695,-48.237,179.272,6.266,149.349
C04923=1132.142,-29.945,-48.225,179.269,6.266,149.350
C04924=1132.146,-30.194,-48.213,179.267,6.265,149.350
C04925=1132.152,-30.444,-48.201,179.265,6.264,149.351
C04926=1132.157,-30.694,-48.189,179.263,6.264,149.351
C04927=1132.162,-30.944,-48.178,179.260,6.263,149.352
C04928=1132.167,-31.194,-48.166,179.258,6.262,149.352
C04929=1132.173,-31.443,-48.155,179.256,6.262,149.353
C04930=1132.178,-31.692,-48.143,179.253,6.261,149.353
C04931=1132.183,-31.942,-48.132,179.251,6.261,149.354
C04932=1132.188,-32.192,-48.120,179.249,6.260,149.354
C04933=1132.193,-32.442,-48.108,179.246,6.259,149.355
C04934=1132.199,-32.692,-48.096,179.244,6.259,149.356
C04935=1132.204,-32.941,-48.086,179.241,6.257,149.356
C04936=1132.210,-33.191,-48.074,179.239,6.256,149.357
C04937=1132.214,-33.440,-48.062,179.236,6.256,149.357
C04938=1132.219,-33.690,-48.050,179.234,6.255,149.358
C04939=1132.225,-33.940,-48.038,179.232,6.254,149.358
C04940=1132.229,-34.189,-48.027,179.230,6.253,149.359
C04941=1132.235,-34.438,-48.015,179.227,6.253,149.359
C04942=1132.240,-34.688,-48.004,179.225,6.252,149.360
C04943=1132.246,-34.938,-47.992,179.222,6.252,149.360
C04944=1132.251,-35.189,-47.981,179.220,6.251,149.361
C04945=1132.256,-35.438,-47.969,179.218,6.250,149.361
C04946=1132.262,-35.687,-47.958,179.215,6.250,149.362
C04947=1132.267,-35.937,-47.947,179.213,6.249,149.362
C04948=1132.272,-36.187,-47.935,179.211,6.248,149.363
C04949=1132.277,-36.437,-47.923,179.208,6.248,149.364
C04950=1132.282,-36.687,-47.912,179.206,6.247,149.364
C04951=1132.288,-36.935,-47.901,179.204,6.246,149.365
C04952=1132.293,-37.185,-47.889,179.201,6.246,149.365
C04953=1132.298,-37.435,-47.877,179.199,6.245,149.366
C04954=1132.303,-37.685,-47.866,179.197,6.244,149.366
C04955=1132.308,-37.934,-47.855,179.194,6.244,149.367
C04956=1132.314,-38.184,-47.844,179.192,6.243,149.367
C04957=1132.319,-38.434,-47.832,179.190,6.242,149.368
C04958=1132.324,-38.684,-47.820,179.188,6.241,149.368
C04959=1132.330,-38.933,-47.809,179.185,6.241,149.369
C04960=1132.335,-39.183,-47.798,179.183,6.240,149.370
C04961=1132.340,-39.432,-47.786,179.181,6.239,149.370
C04962=1132.346,-39.682,-47.775,179.179,6.239,149.370
C04963=1132.351,-39.932,-47.764,179.176,6.238,149.371
C04964=1132.356,-40.182,-47.752,179.174,6.238,149.372
C04965=1132.361,-40.432,-47.741,179.171,6.237,149.372
C04966=1132.367,-40.681,-47.729,179.169,6.236,149.373
C04967=1132.372,-40.930,-47.718,179.167,6.236,149.373
C04968=1132.377,-41.181,-47.707,179.164,6.235,149.374
C04969=1132.383,-41.430,-47.696,179.162,6.234,149.374
C04970=1132.387,-41.679,-47.685,179.160,6.234,149.375
C04971=1132.393,-41.929,-47.673,179.157,6.233,149.375
C04972=1132.398,-42.180,-47.662,179.155,6.232,149.376
C04973=1132.404,-42.429,-47.651,179.153,6.231,149.376
C04974=1132.408,-42.679,-47.639,179.150,6.231,149.377
C04975=1132.413,-42.928,-47.628,179.148,6.230,149.378
C04976=1132.419,-43.178,-47.617,179.147,6.230,149.378
C04977=1132.424,-43.428,-47.606,179.144,6.230,149.379
C04978=1132.430,-43.678,-47.594,179.142,6.229,149.379
C04979=1132.435,-43.927,-47.584,179.140,6.228,149.380
C04980=1132.440,-44.177,-47.573,179.137,6.227,149.380
C04981=1132.445,-44.427,-47.561,179.135,6.227,149.381
C04982=1132.451,-44.676,-47.550,179.133,6.226,149.381
C04983=1132.456,-44.926,-47.539,179.130,6.226,149.382
C04984=1132.461,-45.176,-47.527,179.128,6.225,149.382
C04985=1132.466,-45.425,-47.517,179.125,6.224,149.383
C04986=1132.471,-45.675,-47.506,179.123,6.224,149.383
C04987=1132.477,-45.925,-47.494,179.121,6.223,149.384
C04988=1132.482,-46.174,-47.484,179.119,6.222,149.384
C04989=1132.487,-46.424,-47.473,179.116,6.222,149.385
C04990=1132.493,-46.673,-47.461,179.114,6.221,149.386
C04991=1132.498,-46.924,-47.450,179.112,6.220,149.386
C04992=1132.503,-47.173,-47.439,179.110,6.219,149.387
C04993=1132.508,-47.423,-47.429,179.107,6.219,149.387
C04994=1132.514,-47.673,-47.417,179.105,6.218,149.388
C04995=1132.519,-47.922,-47.406,179.103,6.217,149.388
C04996=1132.524,-48.172,-47.396,179.100,6.217,149.389
C04997=1132.530,-48.422,-47.384,179.098,6.217,149.389
C04998=1132.535,-48.671,-47.374,179.096,6.216,149.390
C04999=1132.540,-48.921,-47.362,179.094,6.216,149.390
C05000=1132.545,-49.170,-47.352,179.092,6.215,149.391
C05001=1132.551,-49.420,-47.340,179.089,6.214,149.392
C05002=1132.556,-49.671,-47.330,179.087,6.214,149.392
C05003=1132.561,-49.920,-47.319,179.085,6.213,149.393
C05004=1132.566,-50.170,-47.308,179.083,6.212,149.393
C05005=1132.572,-50.419,-47.297,179.080,6.212,149.394
C05006=1132.577,-50.690,-47.285,179.078,6.211,149.394
C05007=1132.583,-50.961,-47.273,179.075,6.211,149.395
C05008=1132.589,-51.232,-47.261,179.073,6.210,149.395
C05009=1132.595,-51.503,-47.249,179.071,6.209,149.396
C05010=1132.600,-51.752,-47.239,179.068,6.209,149.397
C05011=1132.605,-52.002,-47.228,179.066,6.208,149.397
C05012=1132.610,-52.252,-47.217,179.064,6.207,149.397
C05013=1132.615,-52.501,-47.206,179.061,6.206,149.398
C05014=1132.620,-52.751,-47.196,179.059,6.206,149.399
C05015=1132.626,-53.000,-47.184,179.057,6.205,149.399
C05016=1132.631,-53.251,-47.174,179.054,6.204,149.400
C05017=1132.637,-53.500,-47.163,179.052,6.204,149.400
C05018=1132.642,-53.750,-47.152,179.050,6.204,149.401
C05019=1132.647,-53.999,-47.142,179.048,6.203,149.401
C05020=1132.652,-54.249,-47.131,179.046,6.202,149.402
C05021=1132.658,-54.499,-47.120,179.044,6.202,149.402
C05022=1132.663,-54.749,-47.109,179.041,6.201,149.403
C05023=1132.669,-54.998,-47.098,179.039,6.201,149.403
C05024=1132.674,-55.248,-47.088,179.036,6.200,149.404
C05025=1132.679,-55.498,-47.077,179.034,6.199,149.404
C05026=1132.684,-55.747,-47.066,179.032,6.198,149.405
C05027=1132.690,-55.997,-47.056,179.029,6.198,149.406
C05028=1132.695,-56.247,-47.045,179.028,6.198,149.406
C05029=1132.700,-56.496,-47.034,179.026,6.197,149.407
C05030=1132.705,-56.746,-47.024,179.023,6.196,149.407
C05031=1132.710,-56.996,-47.014,179.021,6.196,149.408
C05032=1132.716,-57.246,-47.002,179.019,6.195,149.408
C05033=1132.721,-57.495,-46.992,179.016,6.194,149.409
C05034=1132.726,-57.746,-46.981,179.014,6.194,149.409
C05035=1132.732,-57.995,-46.971,179.012,6.193,149.410
C05036=1132.737,-58.245,-46.960,179.010,6.193,149.410
C05037=1132.742,-58.494,-46.949,179.008,6.193,149.411
C05038=1132.747,-58.745,-46.939,179.006,6.192,149.411
C05039=1132.753,-58.994,-46.929,179.003,6.191,149.412
C05040=1132.758,-59.244,-46.917,179.001,6.191,149.413
C05041=1132.763,-59.493,-46.907,178.998,6.190,149.413
C05042=1132.769,-59.743,-46.897,178.996,6.189,149.413
C05043=1132.774,-59.993,-46.886,178.994,6.188,149.414
C05044=1132.779,-60.242,-46.875,178.992,6.189,149.415
C05045=1132.784,-60.492,-46.865,178.990,6.188,149.415
C05046=1132.790,-60.742,-46.855,178.988,6.187,149.416
C05047=1132.795,-60.992,-46.844,178.985,6.186,149.416
C05048=1132.800,-61.242,-46.834,178.983,6.186,149.417
C05049=1132.806,-61.491,-46.824,178.981,6.185,149.417
C05050=1132.811,-61.741,-46.812,178.978,6.185,149.418
C05051=1132.816,-61.990,-46.802,178.977,6.185,149.418
C05052=1132.821,-62.241,-46.791,178.975,6.184,149.419
C05053=1132.827,-62.490,-46.781,178.972,6.183,149.419
C05054=1132.832,-62.740,-46.771,178.970,6.183,149.420
C05055=1132.837,-62.990,-46.760,178.968,6.182,149.420
C05056=1132.843,-63.239,-46.750,178.965,6.181,149.421
C05057=1132.848,-63.489,-46.739,178.963,6.180,149.421
C05058=1132.853,-63.739,-46.729,178.961,6.181,149.422
C05059=1132.858,-63.988,-46.719,178.959,6.180,149.423
C05060=1132.863,-64.238,-46.709,178.957,6.179,149.423
C05061=1132.869,-64.488,-46.698,178.955,6.179,149.424
C05062=1132.874,-64.737,-46.688,178.952,6.178,149.424
C05063=1132.879,-64.987,-46.678,178.950,6.177,149.425
C05064=1132.885,-65.237,-46.667,178.948,6.177,149.425
C05065=1132.890,-65.487,-46.657,178.946,6.177,149.426
C05066=1132.895,-65.737,-46.647,178.944,6.176,149.426
C05067=1132.901,-65.986,-46.636,178.942,6.175,149.427
C05068=1132.906,-66.237,-46.626,178.939,6.175,149.427
C05069=1132.911,-66.486,-46.616,178.937,6.174,149.428
C05070=1132.917,-66.735,-46.606,178.935,6.174,149.428
C05071=1132.922,-66.986,-46.595,178.933,6.173,149.429
C05072=1132.927,-67.235,-46.585,178.931,6.172,149.429
C05073=1132.933,-67.485,-46.575,178.928,6.172,149.430
C05074=1132.938,-67.735,-46.564,178.926,6.171,149.430
C05075=1132.943,-67.984,-46.554,178.924,6.171,149.431
C05076=1132.949,-68.234,-46.544,178.922,6.171,149.431
C05077=1132.954,-68.483,-46.534,178.920,6.170,149.432
C05078=1132.959,-68.733,-46.524,178.917,6.169,149.433
C05079=1132.964,-68.983,-46.514,178.915,6.169,149.433
C05080=1132.970,-69.233,-46.503,178.913,6.168,149.434
C05081=1132.975,-69.483,-46.493,178.911,6.168,149.434
C05082=1132.980,-69.732,-46.483,178.909,6.167,149.435
C05083=1132.985,-69.982,-46.473,178.906,6.167,149.435
C05084=1132.990,-70.232,-46.462,178.904,6.166,149.436
C05085=1132.996,-70.481,-46.452,178.902,6.165,149.436
C05086=1133.002,-70.731,-46.442,178.900,6.165,149.437
C05087=1133.008,-70.981,-46.433,178.898,6.165,149.437
C05088=1133.012,-71.231,-46.423,178.896,6.164,149.438
C05089=1133.017,-71.481,-46.412,178.893,6.163,149.438
C05090=1133.023,-71.730,-46.402,178.891,6.163,149.439
C05091=1133.029,-71.980,-46.392,178.889,6.163,149.439
C05092=1133.033,-72.230,-46.382,178.887,6.162,149.440
C05093=1133.038,-72.479,-46.372,178.885,6.161,149.440
C05094=1133.044,-72.729,-46.362,178.882,6.161,149.441
C05095=1133.050,-72.979,-46.352,178.880,6.160,149.441
C05096=1133.054,-73.229,-46.342,178.879,6.160,149.442
C05097=1133.060,-73.478,-46.332,178.876,6.159,149.442
C05098=1133.065,-73.728,-46.322,178.874,6.159,149.443
C05099=1133.071,-73.977,-46.311,178.872,6.158,149.443
C05100=1133.076,-74.228,-46.302,178.869,6.157,149.444
C05101=1133.081,-74.477,-46.292,178.868,6.158,149.445
C05102=1133.087,-74.727,-46.282,178.866,6.157,149.445
C05103=1133.092,-74.977,-46.272,178.863,6.156,149.446
C05104=1133.098,-75.226,-46.263,178.861,6.155,149.446
C05105=1133.103,-75.477,-46.252,178.859,6.154,149.447
C05106=1133.108,-75.726,-46.242,178.857,6.155,149.447
C05107=1133.113,-75.975,-46.232,178.855,6.154,149.448
C05108=1133.119,-76.226,-46.223,178.853,6.153,149.448
C05109=1133.124,-76.475,-46.213,178.850,6.153,149.449
C05110=1133.130,-76.746,-46.202,178.848,6.152,149.449
C05111=1133.136,-77.019,-46.191,178.846,6.152,149.450
C05112=1133.141,-77.290,-46.180,178.844,6.152,149.450
C05113=1133.147,-77.561,-46.170,178.841,6.151,149.451
C05114=1133.153,-77.811,-46.160,178.839,6.150,149.452
C05115=1133.158,-78.061,-46.149,178.837,6.150,149.452
C05116=1133.163,-78.311,-46.140,178.835,6.149,149.453
C05117=1133.169,-78.560,-46.130,178.833,6.149,149.453
C05118=1133.174,-78.810,-46.120,178.831,6.148,149.453
C05119=1133.179,-79.060,-46.111,178.829,6.147,149.454
C05120=1133.185,-79.309,-46.101,178.826,6.147,149.455
C05121=1133.191,-79.559,-46.091,178.824,6.147,149.455
C05122=1133.195,-79.809,-46.081,178.822,6.146,149.456
C05123=1133.201,-80.059,-46.071,178.820,6.146,149.456
C05124=1133.206,-80.309,-46.062,178.818,6.145,149.457
C05125=1133.211,-80.558,-46.052,178.816,6.145,149.457
C05126=1133.217,-80.808,-46.042,178.814,6.144,149.458
C05127=1133.222,-81.058,-46.033,178.811,6.144,149.458
C05128=1133.227,-81.308,-46.022,178.809,6.143,149.459
C05129=1133.232,-81.557,-46.013,178.808,6.143,149.459
C05130=1133.238,-81.807,-46.003,178.805,6.142,149.460
C05131=1133.243,-82.057,-45.994,178.803,6.141,149.460
C05132=1133.249,-82.307,-45.984,178.801,6.141,149.461
C05133=1133.254,-82.556,-45.974,178.799,6.141,149.461
C05134=1133.260,-82.806,-45.965,178.797,6.140,149.462
C05135=1133.265,-83.056,-45.955,178.795,6.140,149.462
C05136=1133.270,-83.306,-45.946,178.792,6.139,149.463
C05137=1133.275,-83.556,-45.935,178.791,6.139,149.463
C05138=1133.280,-83.805,-45.926,178.789,6.138,149.464
C05139=1133.286,-84.055,-45.916,178.786,6.137,149.464
C05140=1133.291,-84.304,-45.907,178.784,6.137,149.465
C05141=1133.297,-84.555,-45.897,178.782,6.137,149.466
C05142=1133.302,-84.804,-45.887,178.780,6.136,149.466
C05143=1133.308,-85.054,-45.878,178.778,6.136,149.466
C05144=1133.312,-85.303,-45.868,178.776,6.136,149.467
C05145=1133.318,-85.553,-45.859,178.774,6.135,149.467
C05146=1133.323,-85.803,-45.849,178.772,6.134,149.468
C05147=1133.329,-86.053,-45.840,178.769,6.133,149.468
C05148=1133.334,-86.303,-45.831,178.767,6.134,149.469
C05149=1133.339,-86.553,-45.820,178.765,6.133,149.470
C05150=1133.344,-86.803,-45.811,178.763,6.132,149.470
C05151=1133.350,-87.052,-45.801,178.761,6.132,149.471
C05152=1133.355,-87.302,-45.792,178.759,6.132,149.471
C05153=1133.360,-87.551,-45.783,178.757,6.131,149.472
C05154=1133.366,-87.801,-45.773,178.755,6.130,149.472
C05155=1133.371,-88.051,-45.764,178.753,6.130,149.473
C05156=1133.377,-88.301,-45.754,178.751,6.130,149.473
C05157=1133.382,-88.551,-45.745,178.748,6.129,149.474
C05158=1133.387,-88.800,-45.735,178.747,6.129,149.474
C05159=1133.393,-89.050,-45.726,178.745,6.128,149.475
C05160=1133.398,-89.300,-45.717,178.742,6.128,149.475
C05161=1133.403,-89.549,-45.707,178.740,6.127,149.476
C05162=1133.409,-89.799,-45.698,178.739,6.127,149.476
C05163=1133.414,-90.049,-45.688,178.736,6.126,149.477
C05164=1133.419,-90.299,-45.679,178.734,6.125,149.477
C05165=1133.425,-90.549,-45.670,178.732,6.126,149.478
C05166=1133.430,-90.798,-45.660,178.730,6.125,149.478
C05167=1133.435,-91.048,-45.651,178.728,6.124,149.479
C05168=1133.441,-91.298,-45.641,178.726,6.124,149.479
C05169=1133.446,-91.547,-45.632,178.724,6.124,149.480
C05170=1133.451,-91.797,-45.623,178.722,6.123,149.480
C05171=1133.457,-92.047,-45.613,178.720,6.123,149.481
C05172=1133.462,-92.297,-45.604,178.718,6.122,149.481
C05173=1133.467,-92.546,-45.595,178.716,6.121,149.482
C05174=1133.473,-92.797,-45.585,178.714,6.121,149.482
C05175=1133.478,-93.046,-45.577,178.712,6.121,149.483
C05176=1133.483,-93.296,-45.567,178.709,6.120,149.483
C05177=1133.489,-93.546,-45.557,178.707,6.119,149.484
C05178=1133.494,-93.796,-45.549,178.706,6.120,149.484
C05179=1133.499,-94.046,-45.540,178.703,6.119,149.485
C05180=1133.505,-94.295,-45.529,178.701,6.118,149.485
C05181=1133.510,-94.545,-45.521,178.700,6.118,149.486
C05182=1133.515,-94.795,-45.512,178.697,6.117,149.486
C05183=1133.521,-95.045,-45.502,178.695,6.117,149.487
C05184=1133.526,-95.294,-45.493,178.694,6.117,149.487
C05185=1133.531,-95.544,-45.484,178.691,6.116,149.488
C05186=1133.537,-95.794,-45.474,178.689,6.115,149.488
C05187=1133.543,-96.043,-45.466,178.687,6.116,149.489
C05188=1133.548,-96.293,-45.457,178.685,6.115,149.489
C05189=1133.553,-96.542,-45.447,178.683,6.114,149.490
C05190=1133.559,-96.793,-45.438,178.681,6.114,149.490
C05191=1133.564,-97.042,-45.429,178.679,6.113,149.491
C05192=1133.569,-97.292,-45.420,178.677,6.113,149.491
C05193=1133.575,-97.543,-45.410,178.675,6.113,149.492
C05194=1133.580,-97.792,-45.401,178.673,6.112,149.492
C05195=1133.585,-98.042,-45.392,178.671,6.111,149.493
C05196=1133.590,-98.291,-45.383,178.669,6.111,149.493
C05197=1133.596,-98.542,-45.373,178.667,6.110,149.494
C05198=1133.601,-98.791,-45.365,178.665,6.110,149.494
C05199=1133.607,-99.041,-45.356,178.663,6.110,149.495
C05200=1133.612,-99.290,-45.347,178.660,6.109,149.495
C05201=1133.618,-99.541,-45.338,178.659,6.109,149.496
C05202=1133.623,-99.790,-45.329,178.657,6.109,149.496
C05203=1133.628,-100.040,-45.320,178.654,6.108,149.497
C05204=1133.633,-100.290,-45.310,178.653,6.108,149.497
C05205=1133.638,-100.539,-45.301,178.651,6.107,149.498
C05206=1133.644,-100.790,-45.292,178.648,6.106,149.498
C05207=1133.650,-101.039,-45.283,178.647,6.106,149.499
C05208=1133.655,-101.289,-45.274,178.645,6.106,149.499
C05209=1133.660,-101.538,-45.265,178.642,6.105,149.500
C05210=1133.666,-101.788,-45.257,178.641,6.105,149.500
C05211=1133.672,-102.038,-45.247,178.639,6.104,149.501
C05212=1133.677,-102.288,-45.238,178.637,6.103,149.501
C05213=1133.682,-102.538,-45.229,178.635,6.104,149.502
C05214=1133.688,-102.810,-45.220,178.632,6.103,149.503
C05215=1133.694,-103.082,-45.210,178.630,6.102,149.503
C05216=1133.700,-103.354,-45.200,178.628,6.102,149.504
C05217=1133.705,-103.627,-45.191,178.626,6.102,149.504
C05218=1133.711,-103.877,-45.182,178.624,6.101,149.504
C05219=1133.716,-104.127,-45.173,178.622,6.100,149.505
C05220=1133.722,-104.377,-45.164,178.620,6.100,149.505
C05221=1133.727,-104.626,-45.155,178.618,6.100,149.506
C05222=1133.733,-104.876,-45.146,178.616,6.100,149.506
C05223=1133.738,-105.126,-45.137,178.614,6.099,149.507
C05224=1133.743,-105.376,-45.128,178.612,6.099,149.508
C05225=1133.748,-105.625,-45.119,178.610,6.099,149.508
C05226=1133.754,-105.875,-45.111,178.608,6.098,149.509
C05227=1133.759,-106.124,-45.102,178.606,6.097,149.509
C05228=1133.764,-106.374,-45.093,178.604,6.097,149.510
C05229=1133.769,-106.624,-45.084,178.602,6.096,149.510
C05230=1133.774,-106.874,-45.075,178.600,6.096,149.511
C05231=1133.781,-107.123,-45.066,178.598,6.096,149.511
C05232=1133.786,-107.373,-45.057,178.596,6.095,149.512
C05233=1133.792,-107.624,-45.049,178.594,6.095,149.512
C05234=1133.797,-107.874,-45.040,178.592,6.094,149.512
C05235=1133.802,-108.123,-45.031,178.590,6.094,149.513
C05236=1133.808,-108.373,-45.023,178.588,6.093,149.513
C05237=1133.813,-108.622,-45.014,178.586,6.093,149.514
C05238=1133.818,-108.872,-45.005,178.584,6.093,149.514
C05239=1133.823,-109.122,-44.996,178.582,6.092,149.515
C05240=1133.829,-109.371,-44.988,178.581,6.092,149.515
C05241=1133.834,-109.622,-44.979,178.578,6.091,149.516
C05242=1133.840,-109.872,-44.971,178.576,6.091,149.516
C05243=1133.845,-110.121,-44.962,178.575,6.091,149.517
C05244=1133.850,-110.371,-44.953,178.572,6.090,149.517
C05245=1133.856,-110.620,-44.944,178.571,6.090,149.518
C05246=1133.861,-110.871,-44.936,178.569,6.089,149.518
C05247=1133.866,-111.121,-44.927,178.566,6.088,149.519
C05248=1133.872,-111.370,-44.919,178.565,6.088,149.519
C05249=1133.877,-111.620,-44.910,178.563,6.088,149.520
C05250=1133.882,-111.870,-44.901,178.561,6.088,149.520
C05251=1133.888,-112.120,-44.893,178.559,6.087,149.521
C05252=1133.894,-112.369,-44.884,178.557,6.087,149.521
C05253=1133.899,-112.619,-44.875,178.555,6.086,149.522
C05254=1133.904,-112.869,-44.866,178.553,6.086,149.522
C05255=1133.909,-113.119,-44.857,178.551,6.086,149.523
C05256=1133.915,-113.369,-44.850,178.549,6.085,149.523
C05257=1133.920,-113.618,-44.841,178.548,6.085,149.524
C05258=1133.926,-113.868,-44.832,178.545,6.084,149.524
C05259=1133.932,-114.118,-44.824,178.543,6.083,149.525
C05260=1133.937,-114.368,-44.815,178.542,6.084,149.525
C05261=1133.942,-114.618,-44.806,178.539,6.083,149.526
C05262=1133.948,-114.867,-44.798,178.538,6.083,149.526
C05263=1133.953,-115.117,-44.789,178.536,6.082,149.527
C05264=1133.958,-115.367,-44.781,178.534,6.082,149.527
C05265=1133.964,-115.617,-44.772,178.532,6.081,149.528
C05266=1133.969,-115.867,-44.764,178.530,6.081,149.528
C05267=1133.974,-116.116,-44.756,178.528,6.081,149.529
C05268=1133.979,-116.366,-44.747,178.526,6.080,149.529
C05269=1133.985,-116.616,-44.739,178.524,6.080,149.530
C05270=1133.990,-116.866,-44.730,178.522,6.079,149.530
C05271=1133.996,-117.116,-44.721,178.520,6.079,149.530
C05272=1134.002,-117.365,-44.713,178.518,6.079,149.531
C05273=1134.007,-117.615,-44.704,178.517,6.079,149.531
C05274=1134.012,-117.865,-44.695,178.514,6.078,149.532
C05275=1134.018,-118.115,-44.688,178.512,6.077,149.532
C05276=1134.023,-118.365,-44.679,178.511,6.077,149.533
C05277=1134.028,-118.614,-44.671,178.508,6.076,149.533
C05278=1134.034,-118.864,-44.663,178.507,6.076,149.534
C05279=1134.039,-119.114,-44.654,178.505,6.076,149.534
C05280=1134.045,-119.364,-44.646,178.503,6.075,149.535
C05281=1134.050,-119.614,-44.637,178.501,6.075,149.535
C05282=1134.055,-119.863,-44.628,178.500,6.075,149.536
C05283=1134.061,-120.113,-44.621,178.497,6.074,149.536
C05284=1134.066,-120.363,-44.612,178.495,6.073,149.537
C05285=1134.071,-120.613,-44.604,178.494,6.073,149.537
C05286=1134.077,-120.862,-44.595,178.491,6.072,149.538
C05287=1134.083,-121.113,-44.587,178.490,6.073,149.538
C05288=1134.088,-121.362,-44.579,178.488,6.072,149.539
C05289=1134.093,-121.612,-44.571,178.486,6.072,149.539
C05290=1134.098,-121.862,-44.562,178.484,6.071,149.540
C05291=1134.104,-122.111,-44.553,178.482,6.071,149.540
C05292=1134.109,-122.362,-44.545,178.480,6.070,149.541
C05293=1134.115,-122.610,-44.537,178.478,6.070,149.541
C05294=1134.120,-122.861,-44.529,178.476,6.070,149.541
C05295=1134.125,-123.111,-44.520,178.475,6.070,149.542
C05296=1134.131,-123.361,-44.512,178.472,6.069,149.542
C05297=1134.136,-123.610,-44.504,178.470,6.068,149.543
C05298=1134.142,-123.860,-44.496,178.469,6.068,149.543
C05299=1134.147,-124.110,-44.487,178.467,6.067,149.544
C05300=1134.152,-124.360,-44.479,178.465,6.067,149.544
C05301=1134.158,-124.609,-44.471,178.463,6.066,149.545
C05302=1134.163,-124.859,-44.463,178.462,6.067,149.545
C05303=1134.169,-125.109,-44.455,178.459,6.066,149.546
C05304=1134.174,-125.359,-44.446,178.458,6.066,149.546
C05305=1134.180,-125.609,-44.439,178.456,6.065,149.547
C05306=1134.185,-125.858,-44.430,178.454,6.065,149.547
C05307=1134.190,-126.109,-44.422,178.452,6.064,149.548
C05308=1134.196,-126.358,-44.414,178.450,6.064,149.548
C05309=1134.201,-126.609,-44.405,178.448,6.064,149.549
C05310=1134.206,-126.857,-44.397,178.446,6.064,149.549
C05311=1134.212,-127.108,-44.389,178.444,6.063,149.550
C05312=1134.218,-127.358,-44.381,178.443,6.063,149.550
C05313=1134.222,-127.607,-44.373,178.441,6.062,149.550
C05314=1134.228,-127.857,-44.365,178.439,6.062,149.551
C05315=1134.234,-128.107,-44.356,178.437,6.061,149.551
C05316=1134.240,-128.357,-44.349,178.435,6.061,149.552
C05317=1134.244,-128.607,-44.341,178.433,6.061,149.552
C05318=1133.824,-128.618,-44.385,178.430,6.065,149.554
C05319=1133.819,-128.368,-44.393,178.432,6.065,149.554
C05320=1133.813,-128.118,-44.401,178.434,6.065,149.553
C05321=1133.807,-127.868,-44.409,178.435,6.065,149.553
C05322=1133.802,-127.619,-44.417,178.438,6.066,149.552
C05323=1133.797,-127.369,-44.426,178.439,6.066,149.552
C05324=1133.791,-127.119,-44.433,178.441,6.067,149.551
C05325=1133.786,-126.869,-44.442,178.443,6.067,149.551
C05326=1133.780,-126.620,-44.450,178.445,6.067,149.550
C05327=1133.775,-126.369,-44.458,178.447,6.067,149.550
C05328=1133.769,-126.120,-44.466,178.449,6.069,149.549
C05329=1133.764,-125.870,-44.474,178.450,6.068,149.549
C05330=1133.759,-125.620,-44.483,178.452,6.069,149.548
C05331=1133.753,-125.370,-44.491,178.454,6.069,149.548
C05332=1133.748,-125.120,-44.499,178.456,6.070,149.547
C05333=1133.743,-124.871,-44.507,178.458,6.070,149.547
C05334=1133.737,-124.620,-44.515,178.460,6.071,149.546
C05335=1133.731,-124.371,-44.523,178.462,6.071,149.546
C05336=1133.726,-124.121,-44.532,178.464,6.071,149.546
C05337=1133.721,-123.871,-44.540,178.465,6.071,149.545
C05338=1133.715,-123.622,-44.548,178.468,6.072,149.545
C05339=1133.710,-123.372,-44.557,178.470,6.073,149.544
C05340=1133.704,-123.122,-44.564,178.471,6.073,149.544
C05341=1133.700,-122.872,-44.573,178.473,6.074,149.543
C05342=1133.694,-122.622,-44.581,178.475,6.074,149.543
C05343=1133.688,-122.373,-44.589,178.477,6.074,149.542
C05344=1133.683,-122.122,-44.598,178.478,6.074,149.542
C05345=1133.677,-121.873,-44.606,178.481,6.075,149.541
C05346=1133.673,-121.624,-44.614,178.482,6.075,149.541
C05347=1133.667,-121.373,-44.623,178.484,6.076,149.540
C05348=1133.662,-121.124,-44.631,178.486,6.076,149.540
C05349=1133.656,-120.873,-44.639,178.488,6.077,149.539
C05350=1133.650,-120.624,-44.648,178.490,6.077,149.539
C05351=1133.646,-120.374,-44.655,178.492,6.077,149.538
C05352=1133.640,-120.124,-44.664,178.494,6.078,149.538
C05353=1133.634,-119.875,-44.672,178.496,6.078,149.537
C05354=1133.629,-119.625,-44.681,178.498,6.079,149.537
C05355=1133.624,-119.375,-44.690,178.500,6.079,149.536
C05356=1133.618,-119.125,-44.698,178.502,6.079,149.536
C05357=1133.613,-118.875,-44.707,178.503,6.079,149.536
C05358=1133.607,-118.626,-44.714,178.506,6.080,149.535
C05359=1133.602,-118.376,-44.723,178.507,6.080,149.535
C05360=1133.597,-118.126,-44.732,178.509,6.081,149.534
C05361=1133.591,-117.876,-44.740,178.511,6.082,149.534
C05362=1133.586,-117.626,-44.748,178.513,6.082,149.533
C05363=1133.581,-117.377,-44.757,178.515,6.083,149.533
C05364=1133.575,-117.127,-44.765,178.516,6.083,149.532
C05365=1133.569,-116.877,-44.774,178.519,6.083,149.532
C05366=1133.565,-116.627,-44.782,178.520,6.083,149.531
C05367=1133.559,-116.378,-44.790,178.522,6.084,149.531
C05368=1133.554,-116.128,-44.799,178.524,6.084,149.530
C05369=1133.548,-115.877,-44.807,178.526,6.085,149.530
C05370=1133.543,-115.628,-44.816,178.528,6.085,149.529
C05371=1133.537,-115.378,-44.825,178.530,6.085,149.529
C05372=1133.532,-115.129,-44.834,178.532,6.086,149.528
C05373=1133.526,-114.879,-44.841,178.534,6.086,149.528
C05374=1133.521,-114.629,-44.850,178.536,6.087,149.527
C05375=1133.516,-114.379,-44.859,178.538,6.087,149.527
C05376=1133.510,-114.129,-44.867,178.540,6.088,149.526
C05377=1133.505,-113.879,-44.876,178.542,6.088,149.526
C05378=1133.499,-113.630,-44.885,178.544,6.088,149.525
C05379=1133.494,-113.380,-44.894,178.546,6.089,149.525
C05380=1133.488,-113.130,-44.901,178.547,6.089,149.525
C05381=1133.483,-112.880,-44.910,178.550,6.090,149.524
C05382=1133.478,-112.630,-44.919,178.552,6.090,149.524
C05383=1133.473,-112.381,-44.927,178.553,6.090,149.523
C05384=1133.467,-112.131,-44.935,178.556,6.091,149.523
C05385=1133.462,-111.881,-44.944,178.557,6.091,149.522
C05386=1133.457,-111.631,-44.953,178.559,6.092,149.522
C05387=1133.451,-111.382,-44.962,178.561,6.092,149.521
C05388=1133.446,-111.132,-44.971,178.563,6.093,149.521
C05389=1133.441,-110.882,-44.979,178.565,6.093,149.520
C05390=1133.435,-110.632,-44.988,178.567,6.093,149.520
C05391=1133.430,-110.383,-44.996,178.569,6.094,149.519
C05392=1133.424,-110.133,-45.005,178.571,6.094,149.519
C05393=1133.419,-109.883,-45.014,178.573,6.095,149.518
C05394=1133.413,-109.632,-45.023,178.575,6.095,149.518
C05395=1133.407,-109.383,-45.031,178.577,6.095,149.517
C05396=1133.402,-109.133,-45.040,178.579,6.096,149.517
C05397=1133.397,-108.883,-45.049,178.581,6.096,149.516
C05398=1133.392,-108.634,-45.058,178.583,6.097,149.516
C05399=1133.386,-108.384,-45.067,178.585,6.098,149.515
C05400=1133.381,-108.135,-45.075,178.587,6.098,149.515
C05401=1133.375,-107.884,-45.084,178.589,6.098,149.514
C05402=1133.370,-107.634,-45.093,178.590,6.098,149.514
C05403=1133.365,-107.384,-45.101,178.593,6.099,149.513
C05404=1133.359,-107.135,-45.110,178.595,6.100,149.513
C05405=1133.354,-106.885,-45.119,178.596,6.100,149.512
C05406=1133.349,-106.636,-45.128,178.599,6.100,149.512
C05407=1133.344,-106.386,-45.137,178.600,6.100,149.511
C05408=1133.339,-106.136,-45.146,178.602,6.101,149.511
C05409=1133.333,-105.887,-45.154,178.605,6.102,149.510
C05410=1133.328,-105.637,-45.163,178.606,6.102,149.510
C05411=1133.322,-105.387,-45.173,178.608,6.103,149.509
C05412=1133.317,-105.137,-45.181,178.611,6.103,149.509
C05413=1133.311,-104.887,-45.190,178.612,6.103,149.508
C05414=1133.305,-104.637,-45.198,178.615,6.104,149.508
C05415=1133.300,-104.387,-45.207,178.616,6.104,149.507
C05416=1133.295,-104.138,-45.216,178.619,6.104,149.507
C05417=1133.290,-103.888,-45.225,178.621,6.105,149.506
C05418=1133.285,-103.638,-45.234,178.622,6.105,149.506
C05419=1133.279,-103.366,-45.244,178.625,6.106,149.505
C05420=1133.272,-103.094,-45.254,178.627,6.106,149.505
C05421=1133.266,-102.821,-45.263,178.629,6.107,149.504
C05422=1133.261,-102.549,-45.273,178.631,6.107,149.504
C05423=1133.256,-102.299,-45.282,178.633,6.108,149.503
C05424=1133.250,-102.050,-45.291,178.635,6.108,149.503
C05425=1133.245,-101.800,-45.300,178.637,6.108,149.502
C05426=1133.240,-101.550,-45.309,178.639,6.109,149.502
C05427=1133.234,-101.300,-45.318,178.641,6.110,149.501
C05428=1133.228,-101.051,-45.327,178.643,6.110,149.501
C05429=1133.223,-100.801,-45.336,178.645,6.110,149.500
C05430=1133.218,-100.551,-45.345,178.647,6.111,149.500
C05431=1133.213,-100.301,-45.354,178.649,6.111,149.499
C05432=1133.207,-100.051,-45.363,178.651,6.112,149.499
C05433=1133.202,-99.801,-45.372,178.653,6.112,149.498
C05434=1133.197,-99.551,-45.381,178.655,6.113,149.498
C05435=1133.191,-99.303,-45.390,178.657,6.113,149.497
C05436=1133.186,-99.053,-45.399,178.659,6.113,149.497
C05437=1133.180,-98.803,-45.409,178.661,6.114,149.496
C05438=1133.175,-98.553,-45.418,178.663,6.115,149.496
C05439=1133.170,-98.303,-45.426,178.665,6.114,149.495
C05440=1133.165,-98.053,-45.435,178.668,6.115,149.495
C05441=1133.159,-97.803,-45.445,178.670,6.116,149.494
C05442=1133.154,-97.553,-45.454,178.671,6.116,149.494
C05443=1133.149,-97.304,-45.463,178.673,6.117,149.493
C05444=1133.144,-97.054,-45.472,178.676,6.117,149.493
C05445=1133.137,-96.804,-45.481,178.677,6.117,149.492
C05446=1133.132,-96.555,-45.490,178.679,6.118,149.492
C05447=1133.127,-96.305,-45.499,178.682,6.119,149.491
C05448=1133.121,-96.055,-45.509,178.683,6.119,149.491
C05449=1133.116,-95.805,-45.518,178.685,6.120,149.490
C05450=1133.111,-95.556,-45.527,178.688,6.120,149.490
C05451=1133.106,-95.306,-45.536,178.689,6.120,149.489
C05452=1133.100,-95.055,-45.546,178.692,6.121,149.489
C05453=1133.095,-94.806,-45.554,178.694,6.121,149.488
C05454=1133.090,-94.556,-45.564,178.696,6.121,149.488
C05455=1133.084,-94.306,-45.574,178.698,6.122,149.487
C05456=1133.079,-94.056,-45.582,178.700,6.123,149.487
C05457=1133.073,-93.807,-45.591,178.702,6.123,149.486
C05458=1133.068,-93.557,-45.602,178.704,6.124,149.486
C05459=1133.063,-93.307,-45.610,178.706,6.124,149.485
C05460=1133.058,-93.057,-45.619,178.708,6.124,149.485
C05461=1133.052,-92.807,-45.629,178.710,6.125,149.484
C05462=1133.047,-92.558,-45.638,178.712,6.126,149.484
C05463=1133.042,-92.308,-45.647,178.714,6.126,149.483
C05464=1133.036,-92.058,-45.657,178.716,6.126,149.483
C05465=1133.031,-91.809,-45.666,178.719,6.127,149.482
C05466=1133.026,-91.559,-45.675,178.721,6.128,149.482
C05467=1133.020,-91.309,-45.685,178.722,6.128,149.481
C05468=1133.015,-91.059,-45.694,178.725,6.128,149.481
C05469=1133.009,-90.809,-45.704,178.727,6.129,149.480
C05470=1133.004,-90.559,-45.713,178.728,6.129,149.480
C05471=1132.999,-90.310,-45.722,178.731,6.130,149.479
C05472=1132.993,-90.060,-45.732,178.733,6.130,149.479
C05473=1132.988,-89.810,-45.741,178.734,6.130,149.478
C05474=1132.982,-89.561,-45.751,178.737,6.131,149.477
C05475=1132.977,-89.311,-45.760,178.739,6.132,149.477
C05476=1132.972,-89.061,-45.769,178.741,6.132,149.476
C05477=1132.966,-88.811,-45.779,178.743,6.132,149.476
C05478=1132.961,-88.562,-45.788,178.745,6.133,149.476
C05479=1132.956,-88.312,-45.798,178.747,6.134,149.475
C05480=1132.950,-88.062,-45.807,178.749,6.134,149.475
C05481=1132.945,-87.812,-45.816,178.751,6.134,149.474
C05482=1132.940,-87.563,-45.826,178.753,6.135,149.474
C05483=1132.935,-87.313,-45.835,178.755,6.135,149.473
C05484=1132.929,-87.063,-45.845,178.758,6.136,149.472
C05485=1132.924,-86.813,-45.854,178.760,6.136,149.472
C05486=1132.918,-86.564,-45.864,178.762,6.137,149.471
